(* IEC 61131-3 sources: std_i2980_v2.06_cp053/Source/IMM/ieccontrol/ODC1, 23 files *)

(* ---- ABSEInterpreter.pu ---- *)
(*
@h    ! WARNING !
@h    The Kemro K2 system (including software) only meets category B according to EN 954-1,
@h    thus it is not intended for usage in safety-relevant control applications in the field
@h    of personal safety (e.g. emergency stop).
@h    To implement potentially necessary safety-relevant control tasks, always use additional
@h    external safety devices that are intended for the particular purpose, and meet the necessary
@h    functional safety.
@h    For further information see EN 954-1 (EN ISO 13849-1) and/or the K2-x00 user manual, chapter
@h    "CE conformity, directives and standards".

*)

IMPORT_OVER_LISTFILE
 KMEM_HashMapGet
, GET_RUNTIME
, SET_WVEVENT
, cSafetyListLen
, cSEO_END
, cSEO_NOP
, cSEO_START
, cSEO_LD
, cSEO_AND
, cSEO_XOR
, cSEStackSize
, cSEC_BC_EQ_NOT
, cSEC_BC_EQ
, cSEC_BV_EQ_NOT
, cSEC_BV_EQ
, cSEC_RC_GT
, cSEC_RC_LT
, cSEC_RV_GT
, cSEC_RV_LT
, cSEC_POP
, tyMovementRegisterList
, tyODCSequenceInternal
, tsGlbSafetyData
//  tsSafetyCondition
, tySEStack
, tsODCStepPos

END_IMPORT

ALGORITHM_BLOCK ABSEInterpreter #DUMMY_EDIT_BLOCK

SYSTEM_VAR
 sv_MovementsAvailable : tyMovementRegisterList;
 sv_ODCSequenceInt : tyODCSequenceInternal;
 // sv_SafetyCondition : tsSafetyCondition;
END_VAR

SYSTEM_OBJECT
 erSEMovementNotAllowed : ALARM;
END_OBJECT

VAR_EXTERNAL
 g_SafetyData : tsGlbSafetyData;
END_VAR

VAR
 miStackPtr : INT;
 mybStack : tySEStack;
END_VAR

(*
@h    ! WARNING !
@h    The Kemro K2 system (including software) only meets category B according to EN 954-1,
@h    thus it is not intended for usage in safety-relevant control applications in the field
@h    of personal safety (e.g. emergency stop).
@h    To implement potentially necessary safety-relevant control tasks, always use additional
@h    external safety devices that are intended for the particular purpose, and meet the necessary
@h    functional safety.
@h    For further information see EN 954-1 (EN ISO 13849-1) and/or the K2-x00 user manual, chapter
@h    "CE conformity, directives and standards".

*)

FUNCTION fEvaluateCondition : BOOL
 #DUMMY_EDIT_BLOCK

VAR_INPUT
 i : DINT;
END_VAR

VAR_IN_OUT
 bResult : BOOL;
END_VAR
#BEGIN_EDIT_BLOCK
(**************************************** WARNING ********************************************
 *** The KEBA Kemro K2 System including software is not intended for safety control tasks! ***
 ***                       For further information see Comment tab!                        ***
 *********************************************************************************************)

CASE (g_SafetyData.SafetyListTmp[i].Condition) OF
    cSEC_BC_EQ_NOT:
         fEvaluateCondition := g_SafetyData.SafetyListTmp[i].pbParamBool <> EMPTY;
         IF fEvaluateCondition THEN
             bResult := g_SafetyData.SafetyListTmp[i].pbParamBool^ = FALSE;
         END_IF;

    cSEC_BC_EQ:
         fEvaluateCondition := g_SafetyData.SafetyListTmp[i].pbParamBool <> EMPTY;
         IF fEvaluateCondition THEN
             bResult := g_SafetyData.SafetyListTmp[i].pbParamBool^ = TRUE;
         END_IF;

    cSEC_BV_EQ_NOT:
         fEvaluateCondition := (g_SafetyData.SafetyListTmp[i].pbParamBool <> EMPTY)
                        AND (i < cSafetyListLen)
                        AND (g_SafetyData.SafetyListTmp[i+1].pbParamBool <> EMPTY);

         IF fEvaluateCondition THEN
             bResult := g_SafetyData.SafetyListTmp[i].pbParamBool^ <> g_SafetyData.SafetyListTmp[i+1].pbParamBool^;
         END_IF;

    cSEC_BV_EQ:
         fEvaluateCondition := (g_SafetyData.SafetyListTmp[i].pbParamBool <> EMPTY)
                        AND (i < cSafetyListLen)
                        AND (g_SafetyData.SafetyListTmp[i+1].pbParamBool <> EMPTY);

         IF fEvaluateCondition THEN
             bResult := g_SafetyData.SafetyListTmp[i].pbParamBool^ = g_SafetyData.SafetyListTmp[i+1].pbParamBool^;
         END_IF;

    cSEC_RC_GT:
         fEvaluateCondition := (g_SafetyData.SafetyListTmp[i].prParamReal <> EMPTY)
                        AND (i < cSafetyListLen);

         IF fEvaluateCondition THEN
             bResult := g_SafetyData.SafetyListTmp[i].prParamReal^ > g_SafetyData.SafetyListTmp[i+1].rValueReal;
         END_IF;

    cSEC_RC_LT:
         fEvaluateCondition := (g_SafetyData.SafetyListTmp[i].prParamReal <> EMPTY)
                        AND (i < cSafetyListLen);

         IF fEvaluateCondition THEN
             bResult := g_SafetyData.SafetyListTmp[i].prParamReal^ < g_SafetyData.SafetyListTmp[i+1].rValueReal;
         END_IF;

    cSEC_RV_GT:
         fEvaluateCondition := (g_SafetyData.SafetyListTmp[i].prParamReal <> EMPTY)
                        AND (i < cSafetyListLen)
                        AND (g_SafetyData.SafetyListTmp[i+1].prParamReal <> EMPTY);

         IF fEvaluateCondition THEN
             bResult := g_SafetyData.SafetyListTmp[i].prParamReal^ > g_SafetyData.SafetyListTmp[i+1].prParamReal^;
         END_IF;

    cSEC_RV_LT:
         fEvaluateCondition := (g_SafetyData.SafetyListTmp[i].prParamReal <> EMPTY)
                        AND (i < cSafetyListLen)
                        AND (g_SafetyData.SafetyListTmp[i+1].prParamReal <> EMPTY);

         IF fEvaluateCondition THEN
             bResult := g_SafetyData.SafetyListTmp[i].prParamReal^ < g_SafetyData.SafetyListTmp[i+1].prParamReal^;
         END_IF;

    cSEC_POP:
         IF (miStackPtr > 0) THEN
              bResult := mybStack[miStackPtr];
              miStackPtr := miStackPtr - 1;
              fEvaluateCondition := TRUE;
         END_IF;

ELSE
    fEvaluateCondition := FALSE;
END_CASE;

;#END_EDIT_BLOCK END_FUNCTION

(*
@h    ! WARNING !
@h    The Kemro K2 system (including software) only meets category B according to EN 954-1,
@h    thus it is not intended for usage in safety-relevant control applications in the field
@h    of personal safety (e.g. emergency stop).
@h    To implement potentially necessary safety-relevant control tasks, always use additional
@h    external safety devices that are intended for the particular purpose, and meet the necessary
@h    functional safety.
@h    For further information see EN 954-1 (EN ISO 13849-1) and/or the K2-x00 user manual, chapter
@h    "CE conformity, directives and standards".

*)

FUNCTION fRunSafetyCondition : BOOL
 #DUMMY_EDIT_BLOCK

VAR_INPUT
 iIdx : DINT;
END_VAR

VAR
 bValue : BOOL;
 idx : DINT;
 bResult : BOOL;
 bCondition : BOOL;
 bConditionFound : BOOL (* at least one valid condition found *);
END_VAR
#BEGIN_EDIT_BLOCK
(**************************************** WARNING ********************************************
 *** The KEBA Kemro K2 System including software is not intended for safety control tasks! ***
 ***                       For further information see Comment tab!                        ***
 *********************************************************************************************)

bValue := FALSE;
miStackPtr := -1;
idx := iIdx;

bConditionFound := FALSE;
WHILE (idx <= cSafetyListLen) DO
    CASE g_SafetyData.SafetyListTmp[idx].Operator OF
        cSEO_NOP:
            ;

        cSEO_START:
            EXIT;

        cSEO_LD:
            // each LD except first one pushes actual value to stack
            IF (miStackPtr = cSEStackSize) THEN
                bValue := FALSE; // TODO stackoverflow
            END_IF;

            miStackPtr := miStackPtr + 1;

            IF (miStackPtr > 0) THEN
               mybStack[miStackPtr] := bValue;
            END_IF;

            bResult := fEvaluateCondition(idx, bCondition);
            IF bResult THEN
               bValue := bCondition;
            END_IF;

        cSEO_AND:
            bResult := fEvaluateCondition(idx, bCondition);
            IF bResult THEN
                IF miStackPtr >= 0 THEN
                    bValue := bValue AND bCondition;
                ELSE // special case: no "LD" evaluated before, Operator should work like "LD"
                    bValue := bCondition;
                END_IF;
            END_IF;

        cSEO_OR:
            bResult := fEvaluateCondition(idx, bCondition);
            IF bResult THEN
                IF miStackPtr >= 0 THEN
                    bValue := bValue OR bCondition;
                ELSE // special case: no "LD" evaluated before, Operator should work like "LD"
                    bValue := bCondition;
                END_IF;
            END_IF;

        cSEO_XOR:
            bResult := fEvaluateCondition(idx, bCondition);
            IF bResult THEN
                IF miStackPtr >= 0 THEN
                    bValue := bValue XOR bCondition;
                ELSE // special case: no "LD" evaluated before, Operator should work like "LD"
                    bValue := bCondition;
                END_IF;
            END_IF;

        cSEO_END:
            EXIT;
    ELSE
        ; // invalid operation
    END_CASE;

    IF bResult THEN
       bConditionFound := TRUE;
    END_IF;
    idx := idx + 1;
END_WHILE;
//     dummy := Print('ABSEInterpreter.fRunSafetyCondition %s = %d',  sv_SafetyCondition.List[iIdx-1].sParameter, bValue);
fRunSafetyCondition := bValue OR (NOT bConditionFound);

;#END_EDIT_BLOCK END_FUNCTION

(*
@h    ! WARNING !
@h    The Kemro K2 system (including software) only meets category B according to EN 954-1,
@h    thus it is not intended for usage in safety-relevant control applications in the field
@h    of personal safety (e.g. emergency stop).
@h    To implement potentially necessary safety-relevant control tasks, always use additional
@h    external safety devices that are intended for the particular purpose, and meet the necessary
@h    functional safety.
@h    For further information see EN 954-1 (EN ISO 13849-1) and/or the K2-x00 user manual, chapter
@h    "CE conformity, directives and standards".

*)

FUNCTION fCheckMovement : BOOL
 #DUMMY_EDIT_BLOCK

VAR_INPUT
 StepPos : tsODCStepPos (* Step for which dependencies are checked *);
END_VAR

VAR
 i : DINT;
 bAllowed : BOOL;
 iMoveNumber : DINT;
END_VAR
#BEGIN_EDIT_BLOCK
(**************************************** WARNING ********************************************
 *** The KEBA Kemro K2 System including software is not intended for safety control tasks! ***
 ***                       For further information see Comment tab!                        ***
 *********************************************************************************************)

// DBG s:=SET_WVEVENT(1110);
bAllowed := TRUE;

IF (NOT g_SafetyData.bAvailable) THEN
    fCheckMovement := bAllowed;
    RETURN;
END_IF;

iMoveNumber := sv_ODCSequenceInt[StepPos.iColumn][StepPos.iRow].iMoveNumber;

i :=  sv_MovementsAvailable[iMoveNumber].iSESafetyProgIdx;

IF (i > 0) THEN
// DBG    s:=SET_WVEVENT(1112);
    bAllowed := fRunSafetyCondition(i);
// DBG    s:=SET_WVEVENT(1113);
    IF (NOT bAllowed) THEN
       SET_ALARM(Name := erSEMovementNotAllowed,
              SubID1 := sv_MovementsAvailable[iMoveNumber].DeviceId.CompId,
              SubID2 := sv_MovementsAvailable[iMoveNumber].DeviceId.IndexId,
              SubID3 := sv_MovementsAvailable[iMoveNumber].pMovementData^.MoveDir);

    END_IF;
    g_SafetyData.MovementAllowed[sv_MovementsAvailable[iMoveNumber].iODCSafetyMovementsEntry] := bAllowed;
END_IF;

// DBG s:=SET_WVEVENT(1114);

fCheckMovement := bAllowed;

;#END_EDIT_BLOCK END_FUNCTION

END_ALGORITHM_BLOCK

#END_OF_IEC_PART

@Puma @IecEditor 6 113 @Pou 25
@@@BEG_Comment@@@
@h    ! WARNING !
@h    The Kemro K2 system (including software) only meets category B according to EN 954-1,
@h    thus it is not intended for usage in safety-relevant control applications in the field
@h    of personal safety (e.g. emergency stop).
@h    To implement potentially necessary safety-relevant control tasks, always use additional
@h    external safety devices that are intended for the particular purpose, and meet the necessary
@h    functional safety.
@h    For further information see EN 954-1 (EN ISO 13849-1) and/or the K2-x00 user manual, chapter
@h    "CE conformity, directives and standards".

@@@END_Comment@@@

@BEG_Contents

@BEG_Func
@RT(17)FuncTreeContainer
3
@Var @RT(15)KMEM_HashMapGet @RT(0) @T @T @DERIVED 0 @F @RT(22)KEBA_STANDARD_FUNCTION @F
@T
@BEG_Attrib
0 @RT(0) @RT(0)
@END_Attrib
1 1 @F @F @F @F

@Var @RT(11)GET_RUNTIME @RT(0) @T @T @DERIVED 0 @F @RT(22)KEBA_STANDARD_FUNCTION @F
@T
@BEG_Attrib
0 @RT(0) @RT(0)
@END_Attrib
1 1 @F @F @F @F

@Var @RT(11)SET_WVEVENT @RT(0) @T @T @DERIVED 0 @F @RT(22)KEBA_STANDARD_FUNCTION @F
@T
@BEG_Attrib
0 @RT(0) @RT(0)
@END_Attrib
1 1 @F @F @F @F

@END_Func

@BEG_Const
@RT(18)ConstTreeContainer
17
@Var @RT(14)cSafetyListLen @RT(0) @T @F @DT @RT(4)DINT @RT(0) @T @T @BASIC 0 @F
@F @F
@T
@BEG_Attrib
0 @RT(3)200 @RT(39)array length of safety program variable
@END_Attrib
1 1 @F @F @F @F

@Var @RT(8)cSEO_END @RT(0) @T @F @DT @RT(4)UINT @RT(0) @T @T @BASIC 0 @F
@F @F
@T
@BEG_Attrib
0 @RT(5)16#FF @RT(14)END of program
@END_Attrib
1 1 @F @F @F @F

@Var @RT(8)cSEO_NOP @RT(0) @T @F @DT @RT(4)UINT @RT(0) @T @T @BASIC 0 @F
@F @F
@T
@BEG_Attrib
0 @RT(5)16#00 @RT(89)Operator "no operation" (e.g. line contains only additional parameter for last operation)
@END_Attrib
1 1 @F @F @F @F

@Var @RT(10)cSEO_START @RT(0) @T @F @DT @RT(4)UINT @RT(0) @T @T @BASIC 0 @F
@F @F
@T
@BEG_Attrib
0 @RT(5)16#01 @RT(92)start conditions for a certain movement defined in parameter as string (e.g. "Mold1.MoveFwd"
@END_Attrib
1 1 @F @F @F @F

@Var @RT(7)cSEO_LD @RT(0) @T @F @DT @RT(4)UINT @RT(0) @T @T @BASIC 0 @F
@F @F
@T
@BEG_Attrib
0 @RT(5)16#02 @RT(102)Load condition result, if a condition result has been calculated before this result is pushed to stack
@END_Attrib
1 1 @F @F @F @F

@Var @RT(8)cSEO_AND @RT(0) @T @F @DT @RT(4)UINT @RT(0) @T @T @BASIC 0 @F
@F @F
@T
@BEG_Attrib
0 @RT(5)16#03 @RT(53)AND operation with actual result and condition result
@END_Attrib
1 1 @F @F @F @F

@Var @RT(8)cSEO_XOR @RT(0) @T @F @DT @RT(4)UINT @RT(0) @T @T @BASIC 0 @F
@F @F
@T
@BEG_Attrib
0 @RT(5)16#05 @RT(53)XOR operation with actual result and condition result
@END_Attrib
1 1 @F @F @F @F

@Var @RT(12)cSEStackSize @RT(0) @T @F @DT @RT(3)INT @RT(0) @T @T @BASIC 0 @F
@F @F
@T
@BEG_Attrib
0 @RT(1)8 @RT(57)size of stack for condition evaluation in ABSEInterpreter
@END_Attrib
1 1 @F @F @F @F

@Var @RT(14)cSEC_BC_EQ_NOT @RT(0) @T @F @DT @RT(4)UINT @RT(0) @T @T @BASIC 0 @F
@F @F
@T
@BEG_Attrib
0 @RT(5)16#10 @RT(25)Condition BOOL SV = FALSE
@END_Attrib
1 1 @F @F @F @F

@Var @RT(10)cSEC_BC_EQ @RT(0) @T @F @DT @RT(4)UINT @RT(0) @T @T @BASIC 0 @F
@F @F
@T
@BEG_Attrib
0 @RT(5)16#11 @RT(24)Condition BOOL SV = TRUE
@END_Attrib
1 1 @F @F @F @F

@Var @RT(14)cSEC_BV_EQ_NOT @RT(0) @T @F @DT @RT(4)UINT @RT(0) @T @T @BASIC 0 @F
@F @F
@T
@BEG_Attrib
0 @RT(5)16#12 @RT(23)Condition BOOL SV <> SV
@END_Attrib
1 1 @F @F @F @F

@Var @RT(10)cSEC_BV_EQ @RT(0) @T @F @DT @RT(4)UINT @RT(0) @T @T @BASIC 0 @F
@F @F
@T
@BEG_Attrib
0 @RT(5)16#13 @RT(22)Condition BOOL SV = SV
@END_Attrib
1 1 @F @F @F @F

@Var @RT(10)cSEC_RC_GT @RT(0) @T @F @DT @RT(4)UINT @RT(0) @T @T @BASIC 0 @F
@F @F
@T
@BEG_Attrib
0 @RT(5)16#20 @RT(25)Condition REAL SV > VALUE
@END_Attrib
1 1 @F @F @F @F

@Var @RT(10)cSEC_RC_LT @RT(0) @T @F @DT @RT(4)UINT @RT(0) @T @T @BASIC 0 @F
@F @F
@T
@BEG_Attrib
0 @RT(5)16#21 @RT(25)Condition REAL SV < VALUE
@END_Attrib
1 1 @F @F @F @F

@Var @RT(10)cSEC_RV_GT @RT(0) @T @F @DT @RT(4)UINT @RT(0) @T @T @BASIC 0 @F
@F @F
@T
@BEG_Attrib
0 @RT(5)16#22 @RT(22)Condition REAL SV > SV
@END_Attrib
1 1 @F @F @F @F

@Var @RT(10)cSEC_RV_LT @RT(0) @T @F @DT @RT(4)UINT @RT(0) @T @T @BASIC 0 @F
@F @F
@T
@BEG_Attrib
0 @RT(5)16#23 @RT(22)Condition REAL SV < SV
@END_Attrib
1 1 @F @F @F @F

@Var @RT(8)cSEC_POP @RT(0) @T @F @DT @RT(4)UINT @RT(0) @T @T @BASIC 0 @F
@F @F
@T
@BEG_Attrib
0 @RT(5)16#FF @RT(24)pop Condition from Stack
@END_Attrib
1 1 @F @F @F @F

@END_Const

@BEG_Export

@BEG_Kind
@ALGORITHM_BLOCK @RT(15)ABSEInterpreter @STRUCTURED_TEXT
@RT(0) @RT(0) @RT(0)
@END_Kind

@BEG_Dcl
@RT(16)DclTreeContainer
7
@Var @RT(21)sv_MovementsAvailable @RT(0) @T @T @DERIVED 0 @T @T @DT @RT(22)tyMovementRegisterList @RT(0) @T @T @UNKNOWN 0 @F
@F @F
@T
@BEG_Attrib
3 @RT(0) @RT(0) @RT(0)
@END_Attrib
1 8 @F @F @F @F

@Var @RT(17)sv_ODCSequenceInt @RT(0) @T @T @DERIVED 0 @T @T @DT @RT(21)tyODCSequenceInternal @RT(0) @T @T @UNKNOWN 0 @F
@F @F
@T
@BEG_Attrib
3 @RT(0) @RT(0) @RT(0)
@END_Attrib
1 8 @F @F @F @F

@Var @RT(12)g_SafetyData @RT(0) @T @T @DERIVED 0 @T @T @DT @RT(15)tsGlbSafetyData @RT(0) @T @T @UNKNOWN 0 @F
@F @F
@T
@BEG_Attrib
3 @RT(0) @RT(0) @RT(0)
@END_Attrib
1 6 @F @F @F @F

@Var @RT(18)sv_SafetyCondition @RT(0) @T @T @DERIVED 0 @T @T @DT @RT(17)tsSafetyCondition @RT(0) @T @T @UNKNOWN 0 @F
@F @T
@T
@BEG_Attrib
3 @RT(0) @RT(0) @RT(0)
@END_Attrib
1 8 @F @F @F @F

@Var @RT(10)miStackPtr @RT(0) @T @F @DT @RT(3)INT @RT(0) @T @T @BASIC 0 @F
@F @F
@T
@BEG_Attrib
3 @RT(0) @RT(0) @RT(0)
@END_Attrib
1 0 @F @F @F @F

@Var @RT(8)mybStack @RT(0) @T @T @DERIVED 0 @T @T @DT @RT(9)tySEStack @RT(0) @T @T @UNKNOWN 0 @F
@F @F
@T
@BEG_Attrib
3 @RT(0) @RT(0) @RT(0)
@END_Attrib
1 0 @F @F @F @F

@Var @RT(22)erSEMovementNotAllowed @RT(0) @T @F @DT @RT(5)ALARM @RT(0) @T @T @BASIC 0 @F
@F @F
@T
@BEG_Attrib
3 @RT(0) @RT(0) @RT(0)
@END_Attrib
1 7 @F @F @F @F

@END_Dcl

@END_Export

@BEG_Body

3

@BEG_Export

@BEG_Algo
@FUNCTION @RT(18)fEvaluateCondition @STRUCTURED_TEXT
@RT(4)BOOL @RT(0) @RT(0) @F @F
@END_Algo

@BEG_Dcl
@RT(16)DclTreeContainer
2
@Var @RT(1)i @RT(0) @T @F @DT @RT(4)DINT @RT(0) @T @T @BASIC 0 @F
@F @F
@T
@BEG_Attrib
3 @RT(0) @RT(0) @RT(0)
@END_Attrib
1 1 @F @F @F @F

@Var @RT(7)bResult @RT(0) @T @F @DT @RT(4)BOOL @RT(0) @T @T @BASIC 0 @F
@F @F
@T
@BEG_Attrib
3 @RT(0) @RT(0) @RT(0)
@END_Attrib
1 2 @F @F @F @F

@END_Dcl

@END_Export

@BEG_Export

@BEG_Algo
@FUNCTION @RT(19)fRunSafetyCondition @STRUCTURED_TEXT
@RT(4)BOOL @RT(0) @RT(0) @F @F
@END_Algo

@BEG_Dcl
@RT(16)DclTreeContainer
6
@Var @RT(4)iIdx @RT(0) @T @F @DT @RT(4)DINT @RT(0) @T @T @BASIC 0 @F
@F @F
@T
@BEG_Attrib
3 @RT(0) @RT(0) @RT(0)
@END_Attrib
1 1 @F @F @F @F

@Var @RT(6)bValue @RT(0) @T @F @DT @RT(4)BOOL @RT(0) @T @T @BASIC 0 @F
@F @F
@T
@BEG_Attrib
3 @RT(0) @RT(0) @RT(0)
@END_Attrib
1 0 @F @F @F @F

@Var @RT(3)idx @RT(0) @T @F @DT @RT(4)DINT @RT(0) @T @T @BASIC 0 @F
@F @F
@T
@BEG_Attrib
3 @RT(0) @RT(0) @RT(0)
@END_Attrib
1 0 @F @F @F @F

@Var @RT(7)bResult @RT(0) @T @F @DT @RT(4)BOOL @RT(0) @T @T @BASIC 0 @F
@F @F
@T
@BEG_Attrib
3 @RT(0) @RT(0) @RT(0)
@END_Attrib
1 0 @F @F @F @F

@Var @RT(10)bCondition @RT(0) @T @F @DT @RT(4)BOOL @RT(0) @T @T @BASIC 0 @F
@F @F
@T
@BEG_Attrib
3 @RT(0) @RT(0) @RT(0)
@END_Attrib
1 0 @F @F @F @F

@Var @RT(15)bConditionFound @RT(0) @T @F @DT @RT(4)BOOL @RT(0) @T @T @BASIC 0 @F
@F @F
@T
@BEG_Attrib
3 @RT(0) @RT(34)at least one valid condition found @RT(0)
@END_Attrib
1 0 @F @F @F @F

@END_Dcl

@END_Export

@BEG_Export

@BEG_Algo
@FUNCTION @RT(14)fCheckMovement @STRUCTURED_TEXT
@RT(4)BOOL @RT(0) @RT(0) @F @F
@END_Algo

@BEG_Dcl
@RT(16)DclTreeContainer
4
@Var @RT(7)StepPos @RT(0) @T @T @DERIVED 0 @T @T @DT @RT(12)tsODCStepPos @RT(0) @T @T @UNKNOWN 0 @F
@F @F
@T
@BEG_Attrib
3 @RT(0) @RT(39)Step for which dependencies are checked @RT(0)
@END_Attrib
1 1 @F @F @F @F

@Var @RT(1)i @RT(0) @T @F @DT @RT(4)DINT @RT(0) @T @T @BASIC 0 @F
@F @F
@T
@BEG_Attrib
3 @RT(0) @RT(0) @RT(0)
@END_Attrib
1 0 @F @F @F @F

@Var @RT(8)bAllowed @RT(0) @T @F @DT @RT(4)BOOL @RT(0) @T @T @BASIC 0 @F
@F @F
@T
@BEG_Attrib
3 @RT(0) @RT(0) @RT(0)
@END_Attrib
1 0 @F @F @F @F

@Var @RT(11)iMoveNumber @RT(0) @T @F @DT @RT(4)DINT @RT(0) @T @T @BASIC 0 @F
@F @F
@T
@BEG_Attrib
3 @RT(0) @RT(0) @RT(0)
@END_Attrib
1 0 @F @F @F @F

@END_Dcl

@END_Export

@BEG_Body
@TL(86)
(**************************************** WARNING ********************************************
 *** The KEBA Kemro K2 System including software is not intended for safety control tasks! ***
 ***                       For further information see Comment tab!                        ***
 *********************************************************************************************)

CASE (g_SafetyData.SafetyListTmp[i].Condition) OF
    cSEC_BC_EQ_NOT:
         fEvaluateCondition := g_SafetyData.SafetyListTmp[i].pbParamBool <> EMPTY;
         IF fEvaluateCondition THEN
             bResult := g_SafetyData.SafetyListTmp[i].pbParamBool^ = FALSE;
         END_IF;

    cSEC_BC_EQ:
         fEvaluateCondition := g_SafetyData.SafetyListTmp[i].pbParamBool <> EMPTY;
         IF fEvaluateCondition THEN
             bResult := g_SafetyData.SafetyListTmp[i].pbParamBool^ = TRUE;
         END_IF;

    cSEC_BV_EQ_NOT:
         fEvaluateCondition := (g_SafetyData.SafetyListTmp[i].pbParamBool <> EMPTY)
                        AND (i < cSafetyListLen)
                        AND (g_SafetyData.SafetyListTmp[i+1].pbParamBool <> EMPTY);

         IF fEvaluateCondition THEN
             bResult := g_SafetyData.SafetyListTmp[i].pbParamBool^ <> g_SafetyData.SafetyListTmp[i+1].pbParamBool^;
         END_IF;

    cSEC_BV_EQ:
         fEvaluateCondition := (g_SafetyData.SafetyListTmp[i].pbParamBool <> EMPTY)
                        AND (i < cSafetyListLen)
                        AND (g_SafetyData.SafetyListTmp[i+1].pbParamBool <> EMPTY);

         IF fEvaluateCondition THEN
             bResult := g_SafetyData.SafetyListTmp[i].pbParamBool^ = g_SafetyData.SafetyListTmp[i+1].pbParamBool^;
         END_IF;

    cSEC_RC_GT:
         fEvaluateCondition := (g_SafetyData.SafetyListTmp[i].prParamReal <> EMPTY)
                        AND (i < cSafetyListLen);

         IF fEvaluateCondition THEN
             bResult := g_SafetyData.SafetyListTmp[i].prParamReal^ > g_SafetyData.SafetyListTmp[i+1].rValueReal;
         END_IF;

    cSEC_RC_LT:
         fEvaluateCondition := (g_SafetyData.SafetyListTmp[i].prParamReal <> EMPTY)
                        AND (i < cSafetyListLen);

         IF fEvaluateCondition THEN
             bResult := g_SafetyData.SafetyListTmp[i].prParamReal^ < g_SafetyData.SafetyListTmp[i+1].rValueReal;
         END_IF;

    cSEC_RV_GT:
         fEvaluateCondition := (g_SafetyData.SafetyListTmp[i].prParamReal <> EMPTY)
                        AND (i < cSafetyListLen)
                        AND (g_SafetyData.SafetyListTmp[i+1].prParamReal <> EMPTY);

         IF fEvaluateCondition THEN
             bResult := g_SafetyData.SafetyListTmp[i].prParamReal^ > g_SafetyData.SafetyListTmp[i+1].prParamReal^;
         END_IF;

    cSEC_RV_LT:
         fEvaluateCondition := (g_SafetyData.SafetyListTmp[i].prParamReal <> EMPTY)
                        AND (i < cSafetyListLen)
                        AND (g_SafetyData.SafetyListTmp[i+1].prParamReal <> EMPTY);

         IF fEvaluateCondition THEN
             bResult := g_SafetyData.SafetyListTmp[i].prParamReal^ < g_SafetyData.SafetyListTmp[i+1].prParamReal^;
         END_IF;

    cSEC_POP:
         IF (miStackPtr > 0) THEN
              bResult := mybStack[miStackPtr];
              miStackPtr := miStackPtr - 1;
              fEvaluateCondition := TRUE;
         END_IF;

ELSE
    fEvaluateCondition := FALSE;
END_CASE;

@END_Body

@@@BEG_Comment@@@
@TL(12)
@h    ! WARNING !
@h    The Kemro K2 system (including software) only meets category B according to EN 954-1,
@h    thus it is not intended for usage in safety-relevant control applications in the field
@h    of personal safety (e.g. emergency stop).
@h    To implement potentially necessary safety-relevant control tasks, always use additional
@h    external safety devices that are intended for the particular purpose, and meet the necessary
@h    functional safety.
@h    For further information see EN 954-1 (EN ISO 13849-1) and/or the K2-x00 user manual, chapter
@h    "CE conformity, directives and standards".

@@@END_Comment@@@

@BEG_Body
@TL(84)
(**************************************** WARNING ********************************************
 *** The KEBA Kemro K2 System including software is not intended for safety control tasks! ***
 ***                       For further information see Comment tab!                        ***
 *********************************************************************************************)

bValue := FALSE;
miStackPtr := -1;
idx := iIdx;

bConditionFound := FALSE;
WHILE (idx <= cSafetyListLen) DO
    CASE g_SafetyData.SafetyListTmp[idx].Operator OF
        cSEO_NOP:
            ;

        cSEO_START:
            EXIT;

        cSEO_LD:
            // each LD except first one pushes actual value to stack
            IF (miStackPtr = cSEStackSize) THEN
                bValue := FALSE; // TODO stackoverflow
            END_IF;

            miStackPtr := miStackPtr + 1;

            IF (miStackPtr > 0) THEN
               mybStack[miStackPtr] := bValue;
            END_IF;

            bResult := fEvaluateCondition(idx, bCondition);
            IF bResult THEN
               bValue := bCondition;
            END_IF;

        cSEO_AND:
            bResult := fEvaluateCondition(idx, bCondition);
            IF bResult THEN
                IF miStackPtr >= 0 THEN
                    bValue := bValue AND bCondition;
                ELSE // special case: no "LD" evaluated before, Operator should work like "LD"
                    bValue := bCondition;
                END_IF;
            END_IF;

        cSEO_OR:
            bResult := fEvaluateCondition(idx, bCondition);
            IF bResult THEN
                IF miStackPtr >= 0 THEN
                    bValue := bValue OR bCondition;
                ELSE // special case: no "LD" evaluated before, Operator should work like "LD"
                    bValue := bCondition;
                END_IF;
            END_IF;

        cSEO_XOR:
            bResult := fEvaluateCondition(idx, bCondition);
            IF bResult THEN
                IF miStackPtr >= 0 THEN
                    bValue := bValue XOR bCondition;
                ELSE // special case: no "LD" evaluated before, Operator should work like "LD"
                    bValue := bCondition;
                END_IF;
            END_IF;

        cSEO_END:
            EXIT;
    ELSE
        ; // invalid operation
    END_CASE;

    IF bResult THEN
       bConditionFound := TRUE;
    END_IF;
    idx := idx + 1;
END_WHILE;
//     dummy := Print('ABSEInterpreter.fRunSafetyCondition %s = %d',  sv_SafetyCondition.List[iIdx-1].sParameter, bValue);
fRunSafetyCondition := bValue OR (NOT bConditionFound);

@END_Body

@@@BEG_Comment@@@
@TL(12)
@h    ! WARNING !
@h    The Kemro K2 system (including software) only meets category B according to EN 954-1,
@h    thus it is not intended for usage in safety-relevant control applications in the field
@h    of personal safety (e.g. emergency stop).
@h    To implement potentially necessary safety-relevant control tasks, always use additional
@h    external safety devices that are intended for the particular purpose, and meet the necessary
@h    functional safety.
@h    For further information see EN 954-1 (EN ISO 13849-1) and/or the K2-x00 user manual, chapter
@h    "CE conformity, directives and standards".

@@@END_Comment@@@

@BEG_Body
@TL(36)
(**************************************** WARNING ********************************************
 *** The KEBA Kemro K2 System including software is not intended for safety control tasks! ***
 ***                       For further information see Comment tab!                        ***
 *********************************************************************************************)

// DBG s:=SET_WVEVENT(1110);
bAllowed := TRUE;

IF (NOT g_SafetyData.bAvailable) THEN
    fCheckMovement := bAllowed;
    RETURN;
END_IF;

iMoveNumber := sv_ODCSequenceInt[StepPos.iColumn][StepPos.iRow].iMoveNumber;

i :=  sv_MovementsAvailable[iMoveNumber].iSESafetyProgIdx;

IF (i > 0) THEN
// DBG    s:=SET_WVEVENT(1112);
    bAllowed := fRunSafetyCondition(i);
// DBG    s:=SET_WVEVENT(1113);
    IF (NOT bAllowed) THEN
       SET_ALARM(Name := erSEMovementNotAllowed,
              SubID1 := sv_MovementsAvailable[iMoveNumber].DeviceId.CompId,
              SubID2 := sv_MovementsAvailable[iMoveNumber].DeviceId.IndexId,
              SubID3 := sv_MovementsAvailable[iMoveNumber].pMovementData^.MoveDir);

    END_IF;
    g_SafetyData.MovementAllowed[sv_MovementsAvailable[iMoveNumber].iODCSafetyMovementsEntry] := bAllowed;
END_IF;

// DBG s:=SET_WVEVENT(1114);

fCheckMovement := bAllowed;

@END_Body

@@@BEG_Comment@@@
@TL(12)
@h    ! WARNING !
@h    The Kemro K2 system (including software) only meets category B according to EN 954-1,
@h    thus it is not intended for usage in safety-relevant control applications in the field
@h    of personal safety (e.g. emergency stop).
@h    To implement potentially necessary safety-relevant control tasks, always use additional
@h    external safety devices that are intended for the particular purpose, and meet the necessary
@h    functional safety.
@h    For further information see EN 954-1 (EN ISO 13849-1) and/or the K2-x00 user manual, chapter
@h    "CE conformity, directives and standards".

@@@END_Comment@@@
@END_Body

@END_Contents

(* ---- FCreateODCVersion.pu ---- *)
(*
@h    ! WARNING !
@h    The Kemro K2 system (including software) only meets category B according to EN 954-1,
@h    thus it is not intended for usage in safety-relevant control applications in the field
@h    of personal safety (e.g. emergency stop).
@h    To implement potentially necessary safety-relevant control tasks, always use additional
@h    external safety devices that are intended for the particular purpose, and meet the necessary
@h    functional safety.
@h    For further information see EN 954-1 (EN ISO 13849-1) and/or the K2-x00 user manual, chapter
@h    "CE conformity, directives and standards".

this file is automatically created by clearcase makebaseline
and contains versioninformation of component
*)

IMPORT_OVER_LISTFILE
 FWriteComponentVersion

END_IMPORT

FUNCTION FCreateODCVersion : BOOL #DUMMY_EDIT_BLOCK

VAR CONSTANT
 sComponentName : STRING(255) := 'ApplMoldMachineODC';
 iComponentNumber : DINT := 6735;
 sVersionString : STRING(255) := 'ApplMoldMachineODC_01.36';
 iVersionMajor : DINT := 1;
 iVersionMinor : DINT := 36;
END_VAR
#BEGIN_EDIT_BLOCK
(**************************************** WARNING ********************************************
 *** The KEBA Kemro K2 System including software is not intended for safety control tasks! ***
 ***                       For further information see Comment tab!                        ***
 *********************************************************************************************)

FCreateODCVersion := FWriteComponentVersion(
        sComponentName,
        iComponentNumber,
        sVersionString,
        iVersionMajor,
        iVersionMinor
);

;#END_EDIT_BLOCK END_FUNCTION

#END_OF_IEC_PART

@Puma @IecEditor 6 68 @Pou 25
@@@BEG_Comment@@@
@h    ! WARNING !
@h    The Kemro K2 system (including software) only meets category B according to EN 954-1,
@h    thus it is not intended for usage in safety-relevant control applications in the field
@h    of personal safety (e.g. emergency stop).
@h    To implement potentially necessary safety-relevant control tasks, always use additional
@h    external safety devices that are intended for the particular purpose, and meet the necessary
@h    functional safety.
@h    For further information see EN 954-1 (EN ISO 13849-1) and/or the K2-x00 user manual, chapter
@h    "CE conformity, directives and standards".

this file is automatically created by clearcase makebaseline
and contains versioninformation of component
@@@END_Comment@@@

@BEG_Contents

@BEG_Func
@RT(17)FuncTreeContainer
1
@Var @RT(22)FWriteComponentVersion @RT(0) @T @F @DT @RT(0) @RT(0) @T @T @UNKNOWN 0 @F
@F @F
@T
@BEG_Attrib
0 @RT(0) @RT(0)
@END_Attrib
1 1 @F @F @F @F

@END_Func

@BEG_Const
@RT(18)ConstTreeContainer
0
@END_Const

@BEG_Export

@BEG_Kind
@FUNCTION @RT(17)FCreateODCVersion @STRUCTURED_TEXT
@RT(4)BOOL @RT(0) @RT(0)
@END_Kind

@BEG_Dcl
@RT(16)DclTreeContainer
5
@Var @RT(14)sComponentName @RT(0) @T @F @DT @RT(11)STRING(255) @RT(0) @T @T @STRING 0 @F @RT(3)255 @F
@F @F
@T
@BEG_Attrib
3 @RT(20)'ApplMoldMachineODC' @RT(0) @RT(0)
@END_Attrib
1 15 @F @F @F @F

@Var @RT(16)iComponentNumber @RT(0) @T @F @DT @RT(4)DINT @RT(0) @T @T @BASIC 0 @F
@F @F
@T
@BEG_Attrib
3 @RT(4)6735 @RT(0) @RT(0)
@END_Attrib
1 15 @F @F @F @F

@Var @RT(14)sVersionString @RT(0) @T @F @DT @RT(11)STRING(255) @RT(0) @T @T @STRING 0 @F @RT(3)255 @F
@F @F
@T
@BEG_Attrib
3 @RT(26)'ApplMoldMachineODC_01.36' @RT(0) @RT(0)
@END_Attrib
1 15 @F @F @F @F

@Var @RT(13)iVersionMajor @RT(0) @T @F @DT @RT(4)DINT @RT(0) @T @T @BASIC 0 @F
@F @F
@T
@BEG_Attrib
3 @RT(1)1 @RT(0) @RT(0)
@END_Attrib
1 15 @F @F @F @F

@Var @RT(13)iVersionMinor @RT(0) @T @F @DT @RT(4)DINT @RT(0) @T @T @BASIC 0 @F
@F @F
@T
@BEG_Attrib
3 @RT(2)36 @RT(0) @RT(0)
@END_Attrib
1 15 @F @F @F @F

@END_Dcl

@END_Export

@BEG_Body
@TL(13)
(**************************************** WARNING ********************************************
 *** The KEBA Kemro K2 System including software is not intended for safety control tasks! ***
 ***                       For further information see Comment tab!                        ***
 *********************************************************************************************)

FCreateODCVersion := FWriteComponentVersion(
        sComponentName,
        iComponentNumber,
        sVersionString,
        iVersionMajor,
        iVersionMinor
);

@END_Body

@END_Contents

(* ---- FSEMoveIDToValue.pu ---- *)
(*
@h    ! WARNING !
@h    The Kemro K2 system (including software) only meets category B according to EN 954-1,
@h    thus it is not intended for usage in safety-relevant control applications in the field
@h    of personal safety (e.g. emergency stop).
@h    To implement potentially necessary safety-relevant control tasks, always use additional
@h    external safety devices that are intended for the particular purpose, and meet the necessary
@h    functional safety.
@h    For further information see EN 954-1 (EN ISO 13849-1) and/or the K2-x00 user manual, chapter
@h    "CE conformity, directives and standards".

"<FU>.<string movedir>" -> "<FU>.<integer movedir>"
e.g. "Mold1.MoveFwd" -> "Mold1.12"

returns true if no error

*)

IMPORT_OVER_LISTFILE
 cMoveFwd
, cMoveBwd

END_IMPORT

FUNCTION FSEMoveIDToValue : BOOL #DUMMY_EDIT_BLOCK

VAR_IN_OUT
 s : STRING(255) (* movedir definition to be converted *);
END_VAR

VAR
 i : DINT;
 sTmpString : STRING(15);
END_VAR
#BEGIN_EDIT_BLOCK
(**************************************** WARNING ********************************************
 *** The KEBA Kemro K2 System including software is not intended for safety control tasks! ***
 ***                       For further information see Comment tab!                        ***
 *********************************************************************************************)

FSEMoveIDToValue := FALSE;

i := FIND(s, ".");

IF (i = 0) THEN
    RETURN;
END_IF;

sTmpString := RIGHT(s, LEN(s) - i);
s := LEFT(s, i);

IF (sTmpString = "MoveBwd") THEN
    i := cMoveBwd;
ELSIF (sTmpString = "MoveFwd") THEN
    i := cMoveFwd;
ELSE
    RETURN;
END_IF;

s := CONCAT(s, DINT_TO_STRING(i));
FSEMoveIDToValue := TRUE;

;#END_EDIT_BLOCK END_FUNCTION

#END_OF_IEC_PART

@Puma @IecEditor 6 113 @Pou 25
@@@BEG_Comment@@@
@h    ! WARNING !
@h    The Kemro K2 system (including software) only meets category B according to EN 954-1,
@h    thus it is not intended for usage in safety-relevant control applications in the field
@h    of personal safety (e.g. emergency stop).
@h    To implement potentially necessary safety-relevant control tasks, always use additional
@h    external safety devices that are intended for the particular purpose, and meet the necessary
@h    functional safety.
@h    For further information see EN 954-1 (EN ISO 13849-1) and/or the K2-x00 user manual, chapter
@h    "CE conformity, directives and standards".

"<FU>.<string movedir>" -> "<FU>.<integer movedir>"
e.g. "Mold1.MoveFwd" -> "Mold1.12"

returns true if no error

@@@END_Comment@@@

@BEG_Contents

@BEG_Func
@RT(17)FuncTreeContainer
0
@END_Func

@BEG_Const
@RT(18)ConstTreeContainer
2
@Var @RT(8)cMoveFwd @RT(0) @T @F @DT @RT(4)DINT @RT(0) @T @T @BASIC 0 @F
@F @F
@T
@BEG_Attrib
0 @RT(2)12 @RT(16)movement forward
@END_Attrib
1 1 @F @F @F @F

@Var @RT(8)cMoveBwd @RT(0) @T @F @DT @RT(4)DINT @RT(0) @T @T @BASIC 0 @F
@F @F
@T
@BEG_Attrib
0 @RT(2)11 @RT(17)movement backward
@END_Attrib
1 1 @F @F @F @F

@END_Const

@BEG_Export

@BEG_Kind
@FUNCTION @RT(16)FSEMoveIDToValue @STRUCTURED_TEXT
@RT(4)BOOL @RT(0) @RT(0)
@END_Kind

@BEG_Dcl
@RT(16)DclTreeContainer
3
@Var @RT(1)s @RT(0) @T @F @DT @RT(11)STRING(255) @RT(0) @T @T @STRING 0 @F @RT(3)255 @F
@F @F
@T
@BEG_Attrib
3 @RT(0) @RT(34)movedir definition to be converted @RT(0)
@END_Attrib
1 2 @F @F @F @F

@Var @RT(1)i @RT(0) @T @F @DT @RT(4)DINT @RT(0) @T @T @BASIC 0 @F
@F @F
@T
@BEG_Attrib
3 @RT(0) @RT(0) @RT(0)
@END_Attrib
1 0 @F @F @F @F

@Var @RT(10)sTmpString @RT(0) @T @F @DT @RT(10)STRING(15) @RT(0) @T @T @STRING 0 @F @RT(2)15 @F
@F @F
@T
@BEG_Attrib
3 @RT(0) @RT(0) @RT(0)
@END_Attrib
1 0 @F @F @F @F

@END_Dcl

@END_Export

@BEG_Body
@TL(28)
(**************************************** WARNING ********************************************
 *** The KEBA Kemro K2 System including software is not intended for safety control tasks! ***
 ***                       For further information see Comment tab!                        ***
 *********************************************************************************************)

FSEMoveIDToValue := FALSE;

i := FIND(s, ".");

IF (i = 0) THEN
    RETURN;
END_IF;

sTmpString := RIGHT(s, LEN(s) - i);
s := LEFT(s, i);

IF (sTmpString = "MoveBwd") THEN
    i := cMoveBwd;
ELSIF (sTmpString = "MoveFwd") THEN
    i := cMoveFwd;
ELSE
    RETURN;
END_IF;

s := CONCAT(s, DINT_TO_STRING(i));
FSEMoveIDToValue := TRUE;

@END_Body

@END_Contents

(* ---- FBAddDependency.pu ---- *)
IMPORT_OVER_LISTFILE
 tyODCDependencyArray
, tsODCDeviceMovementList
, tyMovementRegisterList

END_IMPORT

FUNCTION_BLOCK FBAddDependency #DUMMY_EDIT_BLOCK

VAR_INPUT
 iFuIndex : DINT (* index in sv_ODCDeviceMovements *);
 iMoveNr : DINT (* 0: not safety relevant, >0: movement number *);
 iCount : DINT;
 iMode : DINT (* 0: replace existing dependency 1: add condition to actual dependency  *);
END_VAR

VAR_IN_OUT
 Dependency : tyODCDependencyArray (* actual step dependency *);
END_VAR

SYSTEM_VAR
 sv_ODCDeviceMovements : tsODCDeviceMovementList (* list of all devices that registered movements for the ODC *);
 sv_MovementsAvailable : tyMovementRegisterList;
END_VAR

VAR_TEMP
 i : DINT;
 k : DINT;
END_VAR

VAR
 tmpDependency : LWORD;
 iInstanceableMovement : DINT;
 iBitNumber : DINT;
END_VAR
#BEGIN_EDIT_BLOCK
(**************************************** WARNING ********************************************
 *** The KEBA Kemro K2 System including software is not intended for safety control tasks! ***
 ***                       For further information see Comment tab!                        ***
 *********************************************************************************************)

IF iMoveNr <= 0 THEN
   Dependency[iFuIndex].Dependency := cNoDependency;
ELSE
   //get movement number in sv_ODCDeviceMovements
   FOR i := 1 TO sv_ODCDeviceMovements.Devices[iFuIndex].iNumberOfMovements DO

      IF sv_ODCDeviceMovements.Devices[iFuIndex].Movements[i]^ = sv_MovementsAvailable[iMoveNr].pMovementData^ THEN
         //move number found -> set the according bit
         tmpDependency := cFirstBit;

         //first movement: shift right 0, second movement: shift right 1, ...
         tmpDependency := SHR(tmpDependency, (i-1));

         IF iMode = 0 THEN
            //replace dependency
            Dependency[iFuIndex].Dependency := tmpDependency;
         ELSE
            //add dependency
            Dependency[iFuIndex].Dependency := Dependency[iFuIndex].Dependency OR tmpDependency;
         END_IF;

         //check if it is an instanceable movement and set correct bit
         IF sv_ODCDeviceMovements.Devices[iFuIndex].Movements[i]^.bInstanceable THEN
            tmpDependency := cFirstBit;

            //first instanceable movement: bit 21-30, second instanceable movement: bit 31-40
            //third instanceable movement: bit 41-50, fourth instanceable movement: bit 51-60

            //find out if it is the first, second, third or fourth instanceable movement in this function unit
            iInstanceableMovement := 1;
            FOR k := 1 TO cMaxSRInstanceableMovements DO
               IF i = sv_ODCDeviceMovements.Devices[iFuIndex].InstanceableMovements[k] THEN
                  iInstanceableMovement := k;
                  EXIT;
               END_IF;
            END_FOR;

            iBitNumber := cMaxDeviceMovements + ((iInstanceableMovement - 1) * cMaxIntermediateConditions) + iCount - 1;
            tmpDependency := SHR(tmpDependency, iBitNumber);

            //mode must not be checked here
            Dependency[iFuIndex].Dependency := Dependency[iFuIndex].Dependency OR tmpDependency;
         END_IF;

         EXIT;
      END_IF;
   END_FOR;
END_IF;

;#END_EDIT_BLOCK END_FUNCTION_BLOCK

#END_OF_IEC_PART

@Puma @IecEditor 6 127 @Pou 25
@@@BEG_Comment@@@

@@@END_Comment@@@

@BEG_Contents

@BEG_Func
@RT(17)FuncTreeContainer
0
@END_Func

@BEG_Const
@RT(18)ConstTreeContainer
0
@END_Const

@BEG_Export

@BEG_Kind
@FUNCTION_BLOCK @RT(15)FBAddDependency @STRUCTURED_TEXT
@RT(0) @RT(0) @RT(0)
@END_Kind

@BEG_Dcl
@RT(16)DclTreeContainer
12
@Var @RT(8)iFuIndex @RT(0) @T @F @DT @RT(4)DINT @RT(0) @T @T @BASIC 0 @F
@F @F
@T
@BEG_Attrib
3 @RT(0) @RT(30)index in sv_ODCDeviceMovements @RT(0)
@END_Attrib
1 1 @F @F @F @F

@Var @RT(7)iMoveNr @RT(0) @T @F @DT @RT(4)DINT @RT(0) @T @T @BASIC 0 @F
@F @F
@T
@BEG_Attrib
3 @RT(0) @RT(43)0: not safety relevant, >0: movement number @RT(0)
@END_Attrib
1 1 @F @F @F @F

@Var @RT(6)iCount @RT(0) @T @F @DT @RT(4)DINT @RT(0) @T @T @BASIC 0 @F
@F @F
@T
@BEG_Attrib
3 @RT(0) @RT(0) @RT(0)
@END_Attrib
1 1 @F @F @F @F

@Var @RT(5)iMode @RT(0) @T @F @DT @RT(4)DINT @RT(0) @T @T @BASIC 0 @F
@F @F
@T
@BEG_Attrib
3 @RT(0) @RT(69)0: replace existing dependency 1: add condition to actual dependency  @RT(0)
@END_Attrib
1 1 @F @F @F @F

@Var @RT(10)Dependency @RT(0) @T @T @DERIVED 0 @T @T @DT @RT(20)tyODCDependencyArray @RT(0) @T @T @UNKNOWN 0 @F
@F @F
@T
@BEG_Attrib
3 @RT(0) @RT(22)actual step dependency @RT(0)
@END_Attrib
1 2 @F @F @F @F

@Var @RT(1)i @RT(0) @T @F @DT @RT(4)DINT @RT(0) @T @T @BASIC 0 @F
@F @F
@T
@BEG_Attrib
3 @RT(0) @RT(0) @RT(0)
@END_Attrib
1 4 @F @F @F @F

@Var @RT(13)tmpDependency @RT(0) @T @F @DT @RT(5)LWORD @RT(0) @T @T @BASIC 0 @F
@F @F
@T
@BEG_Attrib
3 @RT(0) @RT(0) @RT(0)
@END_Attrib
1 0 @F @F @F @F

@Var @RT(21)sv_ODCDeviceMovements @RT(0) @T @T @DERIVED 0 @T @T @DT @RT(23)tsODCDeviceMovementList @RT(0) @T @T @UNKNOWN 0 @F
@F @F
@T
@BEG_Attrib
3 @RT(0) @RT(57)list of all devices that registered movements for the ODC @RT(0)
@END_Attrib
1 8 @F @F @F @F

@Var @RT(21)sv_MovementsAvailable @RT(0) @T @T @DERIVED 0 @T @T @DT @RT(22)tyMovementRegisterList @RT(0) @T @T @UNKNOWN 0 @F
@F @F
@T
@BEG_Attrib
3 @RT(0) @RT(0) @RT(0)
@END_Attrib
1 8 @F @F @F @F

@Var @RT(1)k @RT(0) @T @F @DT @RT(4)DINT @RT(0) @T @T @BASIC 0 @F
@F @F
@T
@BEG_Attrib
3 @RT(0) @RT(0) @RT(0)
@END_Attrib
1 4 @F @F @F @F

@Var @RT(21)iInstanceableMovement @RT(0) @T @F @DT @RT(4)DINT @RT(0) @T @T @BASIC 0 @F
@F @F
@T
@BEG_Attrib
3 @RT(0) @RT(0) @RT(0)
@END_Attrib
1 0 @F @F @F @F

@Var @RT(10)iBitNumber @RT(0) @T @F @DT @RT(4)DINT @RT(0) @T @T @BASIC 0 @F
@F @F
@T
@BEG_Attrib
3 @RT(0) @RT(0) @RT(0)
@END_Attrib
1 0 @F @F @F @F

@END_Dcl

@END_Export

@BEG_Body
@TL(54)
(**************************************** WARNING ********************************************
 *** The KEBA Kemro K2 System including software is not intended for safety control tasks! ***
 ***                       For further information see Comment tab!                        ***
 *********************************************************************************************)

IF iMoveNr <= 0 THEN
   Dependency[iFuIndex].Dependency := cNoDependency;
ELSE
   //get movement number in sv_ODCDeviceMovements
   FOR i := 1 TO sv_ODCDeviceMovements.Devices[iFuIndex].iNumberOfMovements DO

      IF sv_ODCDeviceMovements.Devices[iFuIndex].Movements[i]^ = sv_MovementsAvailable[iMoveNr].pMovementData^ THEN
         //move number found -> set the according bit
         tmpDependency := cFirstBit;

         //first movement: shift right 0, second movement: shift right 1, ...
         tmpDependency := SHR(tmpDependency, (i-1));

         IF iMode = 0 THEN
            //replace dependency
            Dependency[iFuIndex].Dependency := tmpDependency;
         ELSE
            //add dependency
            Dependency[iFuIndex].Dependency := Dependency[iFuIndex].Dependency OR tmpDependency;
         END_IF;

         //check if it is an instanceable movement and set correct bit
         IF sv_ODCDeviceMovements.Devices[iFuIndex].Movements[i]^.bInstanceable THEN
            tmpDependency := cFirstBit;

            //first instanceable movement: bit 21-30, second instanceable movement: bit 31-40
            //third instanceable movement: bit 41-50, fourth instanceable movement: bit 51-60

            //find out if it is the first, second, third or fourth instanceable movement in this function unit
            iInstanceableMovement := 1;
            FOR k := 1 TO cMaxSRInstanceableMovements DO
               IF i = sv_ODCDeviceMovements.Devices[iFuIndex].InstanceableMovements[k] THEN
                  iInstanceableMovement := k;
                  EXIT;
               END_IF;
            END_FOR;

            iBitNumber := cMaxDeviceMovements + ((iInstanceableMovement - 1) * cMaxIntermediateConditions) + iCount - 1;
            tmpDependency := SHR(tmpDependency, iBitNumber);

            //mode must not be checked here
            Dependency[iFuIndex].Dependency := Dependency[iFuIndex].Dependency OR tmpDependency;
         END_IF;

         EXIT;
      END_IF;
   END_FOR;
END_IF;

@END_Body

@END_Contents

(* ---- FBInterpreterCheckIsRightJoin.pu ---- *)
(*
@h    ! WARNING !
@h    The Kemro K2 system (including software) only meets category B according to EN 954-1,
@h    thus it is not intended for usage in safety-relevant control applications in the field
@h    of personal safety (e.g. emergency stop).
@h    To implement potentially necessary safety-relevant control tasks, always use additional
@h    external safety devices that are intended for the particular purpose, and meet the necessary
@h    functional safety.
@h    For further information see EN 954-1 (EN ISO 13849-1) and/or the K2-x00 user manual, chapter
@h    "CE conformity, directives and standards".

Helper for FBInterpreterFindEndOfParalle.pu
Check if we have a join on iLine where the leftmost column with a EndParallel
is iColumnStartBranch
-> this is used to find the end of a parallel branch
*)

IMPORT_OVER_LISTFILE
 cMoveEndParallel
, KODC_Sequence
, FBDebugTrace2

END_IMPORT

FUNCTION_BLOCK FBInterpreterCheckIsRightJoin #DUMMY_EDIT_BLOCK

VAR_IN_OUT
 odcSequence : KODC_Sequence (* [col][line] *);
END_VAR

VAR_INPUT
 iColumnStartBranch : DINT;
 iLine : DINT;
END_VAR

VAR_OUTPUT
 bIsJoin : BOOL;
 bError : BOOL;
END_VAR

VAR_TEMP
 iTmpColumn : DINT;
END_VAR

VAR
 fbDebugTrace2 : FBDebugTrace2;
END_VAR
#BEGIN_EDIT_BLOCK
bError := FALSE;
bIsJoin := FALSE;

FOR iTmpColumn := 1 TO cMaxParallelMovements DO
   IF odcSequence[iTmpColumn][iLine].iMoveId = cMoveEndParallel THEN
      IF iTmpColumn < iColumnStartBranch THEN
         fbDebugTrace2(nODCInterpreter, 'found a EndPParallel at pos:x/x, that tries to join to the wrong parent branch');
         bError := TRUE;
         RETURN; (* error tried to join to somewhere else
                  before we got our wanted join *)
      END_IF;
      IF iTmpColumn = iColumnStartBranch THEN
         (* found where this branch joins again with iColumn *)
         bIsJoin := TRUE;
         RETURN;
      END_IF;
      (* otherwise something else tries to join into this column from the right side
         this is OK, ignore it *)
   END_IF;
END_FOR;

;#END_EDIT_BLOCK END_FUNCTION_BLOCK

#END_OF_IEC_PART

@Puma @IecEditor 6 95 @Pou 25
@@@BEG_Comment@@@
@h    ! WARNING !
@h    The Kemro K2 system (including software) only meets category B according to EN 954-1,
@h    thus it is not intended for usage in safety-relevant control applications in the field
@h    of personal safety (e.g. emergency stop).
@h    To implement potentially necessary safety-relevant control tasks, always use additional
@h    external safety devices that are intended for the particular purpose, and meet the necessary
@h    functional safety.
@h    For further information see EN 954-1 (EN ISO 13849-1) and/or the K2-x00 user manual, chapter
@h    "CE conformity, directives and standards".

Helper for FBInterpreterFindEndOfParalle.pu
Check if we have a join on iLine where the leftmost column with a EndParallel
is iColumnStartBranch
-> this is used to find the end of a parallel branch
@@@END_Comment@@@

@BEG_Contents

@BEG_Func
@RT(17)FuncTreeContainer
0
@END_Func

@BEG_Const
@RT(18)ConstTreeContainer
1
@Var @RT(16)cMoveEndParallel @RT(0) @T @F @DT @RT(0) @RT(0) @T @T @UNKNOWN 0 @F
@F @F
@T
@BEG_Attrib
0 @RT(0) @RT(0)
@END_Attrib
1 1 @F @F @F @F

@END_Const

@BEG_Export

@BEG_Kind
@FUNCTION_BLOCK @RT(29)FBInterpreterCheckIsRightJoin @STRUCTURED_TEXT
@RT(0) @RT(0) @RT(0)
@END_Kind

@BEG_Dcl
@RT(16)DclTreeContainer
7
@Var @RT(11)odcSequence @RT(0) @T @T @DERIVED 0 @T @T @DT @RT(13)KODC_Sequence @RT(0) @T @T @UNKNOWN 0 @F
@F @F
@T
@BEG_Attrib
3 @RT(0) @RT(11)[col][line] @RT(0)
@END_Attrib
1 2 @F @F @F @F

@Var @RT(18)iColumnStartBranch @RT(0) @T @F @DT @RT(4)DINT @RT(0) @T @T @BASIC 0 @F
@F @F
@T
@BEG_Attrib
3 @RT(0) @RT(0) @RT(0)
@END_Attrib
1 1 @F @F @F @F

@Var @RT(5)iLine @RT(0) @T @F @DT @RT(4)DINT @RT(0) @T @T @BASIC 0 @F
@F @F
@T
@BEG_Attrib
3 @RT(0) @RT(0) @RT(0)
@END_Attrib
1 1 @F @F @F @F

@Var @RT(7)bIsJoin @RT(0) @T @F @DT @RT(4)BOOL @RT(0) @T @T @BASIC 0 @F
@F @F
@T
@BEG_Attrib
3 @RT(0) @RT(0) @RT(0)
@END_Attrib
1 3 @F @F @F @F

@Var @RT(6)bError @RT(0) @T @F @DT @RT(4)BOOL @RT(0) @T @T @BASIC 0 @F
@F @F
@T
@BEG_Attrib
3 @RT(0) @RT(0) @RT(0)
@END_Attrib
1 3 @F @F @F @F

@Var @RT(10)iTmpColumn @RT(0) @T @F @DT @RT(4)DINT @RT(0) @T @T @BASIC 0 @F
@F @F
@T
@BEG_Attrib
3 @RT(0) @RT(0) @RT(0)
@END_Attrib
1 4 @F @F @F @F

@Var @RT(13)fbDebugTrace2 @RT(0) @T @T @DERIVED 0 @T @T @DT @RT(13)FBDebugTrace2 @RT(0) @T @T @UNKNOWN 0 @F
@F @F
@T
@BEG_Attrib
3 @RT(0) @RT(0) @RT(0)
@END_Attrib
1 0 @F @F @F @F

@END_Dcl

@END_Export

@BEG_Body
@TL(21)
bError := FALSE;
bIsJoin := FALSE;

FOR iTmpColumn := 1 TO cMaxParallelMovements DO
   IF odcSequence[iTmpColumn][iLine].iMoveId = cMoveEndParallel THEN
      IF iTmpColumn < iColumnStartBranch THEN
         fbDebugTrace2(nODCInterpreter, 'found a EndPParallel at pos:x/x, that tries to join to the wrong parent branch');
         bError := TRUE;
         RETURN; (* error tried to join to somewhere else
                  before we got our wanted join *)
      END_IF;
      IF iTmpColumn = iColumnStartBranch THEN
         (* found where this branch joins again with iColumn *)
         bIsJoin := TRUE;
         RETURN;
      END_IF;
      (* otherwise something else tries to join into this column from the right side
         this is OK, ignore it *)
   END_IF;
END_FOR;

@END_Body

@END_Contents
@@@BEG_Password@@@
NGhzZm9kYzQ=
@@@END_Password@@@

(* ---- FBInterpreterFindEndOfParallel.pu ---- *)
(*
@h    ! WARNING !
@h    The Kemro K2 system (including software) only meets category B according to EN 954-1,
@h    thus it is not intended for usage in safety-relevant control applications in the field
@h    of personal safety (e.g. emergency stop).
@h    To implement potentially necessary safety-relevant control tasks, always use additional
@h    external safety devices that are intended for the particular purpose, and meet the necessary
@h    functional safety.
@h    For further information see EN 954-1 (EN ISO 13849-1) and/or the K2-x00 user manual, chapter
@h    "CE conformity, directives and standards".

Find the end of a parallel branch in
*)

IMPORT_OVER_LISTFILE
 cMoveEndParallel
, FBInterpreterCheckIsRightJoin
, FBDebugTrace2
, KODC_Sequence

END_IMPORT

FUNCTION_BLOCK FBInterpreterFindEndOfParallel #DUMMY_EDIT_BLOCK

VAR_IN_OUT
 odcSequence : KODC_Sequence (* [col][line] *);
END_VAR

VAR_INPUT
 iColumn : DINT;
 iLine : DINT;
END_VAR

VAR_OUTPUT
 iMaxLineOfBranch : DINT;
END_VAR

VAR_TEMP
 i : DINT;
 k : DINT;
END_VAR

VAR
 fbInterpreterCheckIsRightJoin : FBInterpreterCheckIsRightJoin;
 fbDebugTrace2 : FBDebugTrace2;
END_VAR
#BEGIN_EDIT_BLOCK

(* col/line  point to a SP (leftmost of them)*)

iMaxLineOfBranch := 0;

FOR i := 1 TO cMaxParallelMovements DO
   IF odcSequence[i][iLine].iMoveId = cMoveStartParallel THEN
      IF i < iColumn THEN
         fbDebugTrace2(nODCInterpreter, 'error block called wrong iColumn must be the leftmost SP');
         RETURN;
      ELSIF i > iColumn THEN
         (* iColumn itself is skipped since it's join point is the same as at least another join point*)
         FOR k := iLine + 1 TO cMaxODCSteps DO
            IF odcSequence[i][k].iMoveId = cMoveEndParallel THEN
               (* now look to the left if the left most column is
               the same where the parallel branch started *)
               fbInterpreterCheckIsRightJoin(odcSequence := odcSequence, iColumnStartBranch := iColumn, iLine := k);
               IF fbInterpreterCheckIsRightJoin.bIsJoin THEN
                  iMaxLineOfBranch := MAX(iMaxLineOfBranch, k);
                  EXIT;
               END_IF;
               IF fbInterpreterCheckIsRightJoin.bError THEN
                  (* error printed inside the block already *)
                  iMaxLineOfBranch := 0;
                  RETURN;
               END_IF;
            END_IF;
         END_FOR;
      END_IF; // i < iColumn
   END_IF; // odcSequence[i][iLine].iMoveId = cMoveStartParallel
END_FOR;

IF iMaxLineOfBranch = 0 THEN
   fbDebugTrace2(nODCInterpreter, 'no branch join point found????');
   (* error no branch join point found for this branch?? *)
   RETURN;
END_IF;

;#END_EDIT_BLOCK END_FUNCTION_BLOCK

#END_OF_IEC_PART

@Puma @IecEditor 6 95 @Pou 25
@@@BEG_Comment@@@
@h    ! WARNING !
@h    The Kemro K2 system (including software) only meets category B according to EN 954-1,
@h    thus it is not intended for usage in safety-relevant control applications in the field
@h    of personal safety (e.g. emergency stop).
@h    To implement potentially necessary safety-relevant control tasks, always use additional
@h    external safety devices that are intended for the particular purpose, and meet the necessary
@h    functional safety.
@h    For further information see EN 954-1 (EN ISO 13849-1) and/or the K2-x00 user manual, chapter
@h    "CE conformity, directives and standards".

Find the end of a parallel branch in
@@@END_Comment@@@

@BEG_Contents

@BEG_Func
@RT(17)FuncTreeContainer
0
@END_Func

@BEG_Const
@RT(18)ConstTreeContainer
1
@Var @RT(16)cMoveEndParallel @RT(0) @T @F @DT @RT(0) @RT(0) @T @T @UNKNOWN 0 @F
@F @F
@T
@BEG_Attrib
0 @RT(0) @RT(0)
@END_Attrib
1 1 @F @F @F @F

@END_Const

@BEG_Export

@BEG_Kind
@FUNCTION_BLOCK @RT(30)FBInterpreterFindEndOfParallel @STRUCTURED_TEXT
@RT(0) @RT(0) @RT(0)
@END_Kind

@BEG_Dcl
@RT(16)DclTreeContainer
8
@Var @RT(29)fbInterpreterCheckIsRightJoin @RT(0) @T @T @DERIVED 0 @T @T @DT @RT(29)FBInterpreterCheckIsRightJoin @RT(0) @T @T @UNKNOWN 0 @F
@F @F
@T
@BEG_Attrib
3 @RT(0) @RT(0) @RT(0)
@END_Attrib
1 0 @F @F @F @F

@Var @RT(13)fbDebugTrace2 @RT(0) @T @T @DERIVED 0 @T @T @DT @RT(13)FBDebugTrace2 @RT(0) @T @T @UNKNOWN 0 @F
@F @F
@T
@BEG_Attrib
3 @RT(0) @RT(0) @RT(0)
@END_Attrib
1 0 @F @F @F @F

@Var @RT(11)odcSequence @RT(0) @T @T @DERIVED 0 @T @T @DT @RT(13)KODC_Sequence @RT(0) @T @T @UNKNOWN 0 @F
@F @F
@T
@BEG_Attrib
3 @RT(0) @RT(11)[col][line] @RT(0)
@END_Attrib
1 2 @F @F @F @F

@Var @RT(7)iColumn @RT(0) @T @F @DT @RT(4)DINT @RT(0) @T @T @BASIC 0 @F
@F @F
@T
@BEG_Attrib
3 @RT(0) @RT(0) @RT(0)
@END_Attrib
1 1 @F @F @F @F

@Var @RT(5)iLine @RT(0) @T @F @DT @RT(4)DINT @RT(0) @T @T @BASIC 0 @F
@F @F
@T
@BEG_Attrib
3 @RT(0) @RT(0) @RT(0)
@END_Attrib
1 1 @F @F @F @F

@Var @RT(16)iMaxLineOfBranch @RT(0) @T @F @DT @RT(4)DINT @RT(0) @T @T @BASIC 0 @F
@F @F
@T
@BEG_Attrib
3 @RT(0) @RT(0) @RT(0)
@END_Attrib
1 3 @F @F @F @F

@Var @RT(1)i @RT(0) @T @F @DT @RT(4)DINT @RT(0) @T @T @BASIC 0 @F
@F @F
@T
@BEG_Attrib
3 @RT(0) @RT(0) @RT(0)
@END_Attrib
1 4 @F @F @F @F

@Var @RT(1)k @RT(0) @T @F @DT @RT(4)DINT @RT(0) @T @T @BASIC 0 @F
@F @F
@T
@BEG_Attrib
3 @RT(0) @RT(0) @RT(0)
@END_Attrib
1 4 @F @F @F @F

@END_Dcl

@END_Export

@BEG_Body
@TL(39)

(* col/line  point to a SP (leftmost of them)*)

iMaxLineOfBranch := 0;

FOR i := 1 TO cMaxParallelMovements DO
   IF odcSequence[i][iLine].iMoveId = cMoveStartParallel THEN
      IF i < iColumn THEN
         fbDebugTrace2(nODCInterpreter, 'error block called wrong iColumn must be the leftmost SP');
         RETURN;
      ELSIF i > iColumn THEN
         (* iColumn itself is skipped since it's join point is the same as at least another join point*)
         FOR k := iLine + 1 TO cMaxODCSteps DO
            IF odcSequence[i][k].iMoveId = cMoveEndParallel THEN
               (* now look to the left if the left most column is
               the same where the parallel branch started *)
               fbInterpreterCheckIsRightJoin(odcSequence := odcSequence, iColumnStartBranch := iColumn, iLine := k);
               IF fbInterpreterCheckIsRightJoin.bIsJoin THEN
                  iMaxLineOfBranch := MAX(iMaxLineOfBranch, k);
                  EXIT;
               END_IF;
               IF fbInterpreterCheckIsRightJoin.bError THEN
                  (* error printed inside the block already *)
                  iMaxLineOfBranch := 0;
                  RETURN;
               END_IF;
            END_IF;
         END_FOR;
      END_IF; // i < iColumn
   END_IF; // odcSequence[i][iLine].iMoveId = cMoveStartParallel
END_FOR;

IF iMaxLineOfBranch = 0 THEN
   fbDebugTrace2(nODCInterpreter, 'no branch join point found????');
   (* error no branch join point found for this branch?? *)
   RETURN;
END_IF;

@END_Body

@END_Contents
@@@BEG_Password@@@
NGhzZm9kYzQ=
@@@END_Password@@@

(* ---- FBMoveDescription.pu ---- *)
IMPORT_OVER_LISTFILE
 tyMovementRegisterList
, tsODCDeviceMovementList

END_IMPORT

FUNCTION_BLOCK FBMoveDescription #DUMMY_EDIT_BLOCK

VAR_OUTPUT
 sDescription : STRING(255);
END_VAR

VAR_INPUT
 iMoveNr : DINT;
END_VAR

SYSTEM_VAR
 sv_MovementsAvailable : tyMovementRegisterList;
 sv_ODCDeviceMovements : tsODCDeviceMovementList;
END_VAR
#BEGIN_EDIT_BLOCK
(**************************************** WARNING ********************************************
 *** The KEBA Kemro K2 System including software is not intended for safety control tasks! ***
 ***                       For further information see Comment tab!                        ***
 *********************************************************************************************)

sDescription := CONCAT(sv_ODCDeviceMovements.Devices[sv_MovementsAvailable[iMoveNr].iFuIndex].sFuName,
                       " ",
                       sv_MovementsAvailable[iMoveNr].pMovementData^.sMoveId);

;#END_EDIT_BLOCK END_FUNCTION_BLOCK

#END_OF_IEC_PART

@Puma @IecEditor 6 96 @Pou 25
@@@BEG_Comment@@@

@@@END_Comment@@@

@BEG_Contents

@BEG_Func
@RT(17)FuncTreeContainer
0
@END_Func

@BEG_Const
@RT(18)ConstTreeContainer
0
@END_Const

@BEG_Export

@BEG_Kind
@FUNCTION_BLOCK @RT(17)FBMoveDescription @STRUCTURED_TEXT
@RT(0) @RT(0) @RT(0)
@END_Kind

@BEG_Dcl
@RT(16)DclTreeContainer
4
@Var @RT(12)sDescription @RT(0) @T @F @DT @RT(11)STRING(255) @RT(0) @T @T @STRING 0 @F @RT(3)255 @F
@F @F
@T
@BEG_Attrib
3 @RT(0) @RT(0) @RT(0)
@END_Attrib
1 3 @F @F @F @F

@Var @RT(7)iMoveNr @RT(0) @T @F @DT @RT(4)DINT @RT(0) @T @T @BASIC 0 @F
@F @F
@T
@BEG_Attrib
3 @RT(0) @RT(0) @RT(0)
@END_Attrib
1 1 @F @F @F @F

@Var @RT(21)sv_MovementsAvailable @RT(0) @T @T @DERIVED 0 @T @T @DT @RT(22)tyMovementRegisterList @RT(0) @T @T @UNKNOWN 0 @F
@F @F
@T
@BEG_Attrib
3 @RT(0) @RT(0) @RT(0)
@END_Attrib
1 8 @F @F @F @F

@Var @RT(21)sv_ODCDeviceMovements @RT(0) @T @T @RENAMED 0 @T @T @DT @RT(23)tsODCDeviceMovementList @RT(0) @T @T @UNKNOWN 0 @F
@F @F
@T
@BEG_Attrib
3 @RT(0) @RT(0) @RT(0)
@END_Attrib
1 8 @F @F @F @F

@END_Dcl

@END_Export

@BEG_Body
@TL(11)
(**************************************** WARNING ********************************************
 *** The KEBA Kemro K2 System including software is not intended for safety control tasks! ***
 ***                       For further information see Comment tab!                        ***
 *********************************************************************************************)

sDescription := CONCAT(sv_ODCDeviceMovements.Devices[sv_MovementsAvailable[iMoveNr].iFuIndex].sFuName,
                       " ",
                       sv_MovementsAvailable[iMoveNr].pMovementData^.sMoveId);

@END_Body

@END_Contents
@@@BEG_Password@@@
NGhzZm9kYzQ=
@@@END_Password@@@

(* ---- FBSetStepState.pu ---- *)
(*
Update the current state of a step to the internal ODC sequence array
at sv_ODCSequenceInt.StepState

This state is used on the HMI to display errors, the currently executing step
and finished steps.
*)

IMPORT_OVER_LISTFILE
 tyODCSequenceInternal
, tsODCStepPos
, tnODCStepState

END_IMPORT

FUNCTION_BLOCK FBSetStepState #DUMMY_EDIT_BLOCK

VAR_INPUT
 StepPos : tsODCStepPos (* Position of the step for which to update the state *);
 StepState : tnODCStepState (* New state *);
END_VAR

SYSTEM_VAR
 sv_ODCSequenceInt : tyODCSequenceInternal;
END_VAR
#BEGIN_EDIT_BLOCK
(**************************************** WARNING ********************************************
 *** The KEBA Kemro K2 System including software is not intended for safety control tasks! ***
 ***                       For further information see Comment tab!                        ***
 *********************************************************************************************)

sv_ODCSequenceInt[StepPos.iColumn][StepPos.iRow].StepState := StepState;

sv_ODCSequenceInt[StepPos.iColumn][StepPos.iRow].bStepActive := (StepState = nStateActive);
sv_ODCSequenceInt[StepPos.iColumn][StepPos.iRow].bStepDone := (StepState = nStateReady);

;#END_EDIT_BLOCK END_FUNCTION_BLOCK

#END_OF_IEC_PART

@Puma @IecEditor 6 96 @Pou 25
@@@BEG_Comment@@@
Update the current state of a step to the internal ODC sequence array
at sv_ODCSequenceInt.StepState

This state is used on the HMI to display errors, the currently executing step
and finished steps.
@@@END_Comment@@@

@BEG_Contents

@BEG_Func
@RT(17)FuncTreeContainer
0
@END_Func

@BEG_Const
@RT(18)ConstTreeContainer
0
@END_Const

@BEG_Export

@BEG_Kind
@FUNCTION_BLOCK @RT(14)FBSetStepState @STRUCTURED_TEXT
@RT(0) @RT(0) @RT(0)
@END_Kind

@BEG_Dcl
@RT(16)DclTreeContainer
3
@Var @RT(17)sv_ODCSequenceInt @RT(0) @T @T @DERIVED 0 @F @RT(21)tyODCSequenceInternal @F
@T
@BEG_Attrib
3 @RT(0) @RT(0) @RT(0)
@END_Attrib
1 8 @F @F @F @F

@Var @RT(7)StepPos @RT(0) @T @T @DERIVED 0 @T @T @DT @RT(12)tsODCStepPos @RT(0) @T @T @UNKNOWN 0 @F
@F @F
@T
@BEG_Attrib
3 @RT(0) @RT(50)Position of the step for which to update the state @RT(0)
@END_Attrib
1 1 @F @F @F @F

@Var @RT(9)StepState @RT(0) @T @T @DERIVED 0 @T @T @DT @RT(14)tnODCStepState @RT(0) @T @T @UNKNOWN 0 @F
@F @F
@T
@BEG_Attrib
3 @RT(0) @RT(9)New state @RT(0)
@END_Attrib
1 1 @F @F @F @F

@END_Dcl

@END_Export

@BEG_Body
@TL(10)
(**************************************** WARNING ********************************************
 *** The KEBA Kemro K2 System including software is not intended for safety control tasks! ***
 ***                       For further information see Comment tab!                        ***
 *********************************************************************************************)

sv_ODCSequenceInt[StepPos.iColumn][StepPos.iRow].StepState := StepState;

sv_ODCSequenceInt[StepPos.iColumn][StepPos.iRow].bStepActive := (StepState = nStateActive);
sv_ODCSequenceInt[StepPos.iColumn][StepPos.iRow].bStepDone := (StepState = nStateReady);

@END_Body

@END_Contents
@@@BEG_Password@@@
NGhzZm9kYzQ=
@@@END_Password@@@

(* ---- FBStartedMovementAdder.pu ---- *)
(*
@h    ! WARNING !
@h    The Kemro K2 system (including software) only meets category B according to EN 954-1,
@h    thus it is not intended for usage in safety-relevant control applications in the field
@h    of personal safety (e.g. emergency stop).
@h    To implement potentially necessary safety-relevant control tasks, always use additional
@h    external safety devices that are intended for the particular purpose, and meet the necessary
@h    functional safety.
@h    For further information see EN 954-1 (EN ISO 13849-1) and/or the K2-x00 user manual, chapter
@h    "CE conformity, directives and standards".
*)

IMPORT_OVER_LISTFILE
 SET_ALARM
, ASSERT
, cMaxActiveMovements
, tsDeviceId
, tsODCStepPos
, tMoveIdent
, tsStartedMoveDataODCExtended
, KRTOS_Semaphore
, KRTOS_Status
, tsTraceLevel

END_IMPORT

FUNCTION_BLOCK FBStartedMovementAdder #DUMMY_EDIT_BLOCK

VAR_INPUT
 DeviceId : tsDeviceId;
 StepPos : tsODCStepPos;
 MoveId : tMoveIdent;
 MoveDir : tMoveIdent;
 iInstance : DINT;
END_VAR

VAR_OUTPUT
 bOK : BOOL;
END_VAR

SYSTEM_VAR
 sv_StartedManualMovements : tsStartedMoveDataODCExtended;
 sv_TraceLevel : tsTraceLevel;
END_VAR

SYSTEM_OBJECT
 erMaxStartedMovementsExceeded : ALARM;
 erAssert : ALARM;
END_OBJECT

VAR_EXTERNAL
 MovementsSema : KRTOS_Semaphore (* protects sv_StartedManualMovements *);
END_VAR

VAR_TEMP
 i : DINT;
END_VAR

VAR
 dummy : DINT;
 dummy2 : BOOL;
 Status : KRTOS_Status;
END_VAR
#BEGIN_EDIT_BLOCK
(**************************************** WARNING ********************************************
 *** The KEBA Kemro K2 System including software is not intended for safety control tasks! ***
 ***                       For further information see Comment tab!                        ***
 *********************************************************************************************)

bOK := FALSE;

Status := MovementsSema.Wait(WaitTime := cTimeOutSempahore);
IF Status <> KRTOS_Status_OK THEN
   dummy2 := ASSERT(FALSE, erAssert);
   RETURN;
END_IF;

IF sv_StartedManualMovements.iStartedMovements < cMaxActiveMovements THEN
   //add movement to sv_StartedManualMovements
   IF sv_TraceLevel.bODCInterpreter THEN
      dummy := Print('adding started manual movement %d.%d %d/%d pos: %d/%d', DeviceId.CompId, DeviceId.IndexId, MoveId, MoveDir, StepPos.iColumn, StepPos.iRow);
   END_IF;

   sv_StartedManualMovements.iStartedMovements := sv_StartedManualMovements.iStartedMovements +1;
   sv_StartedManualMovements.MoveData[sv_StartedManualMovements.iStartedMovements].DeviceId := DeviceId;
   sv_StartedManualMovements.MoveData[sv_StartedManualMovements.iStartedMovements].MoveDir := MoveDir;
   sv_StartedManualMovements.MoveData[sv_StartedManualMovements.iStartedMovements].MoveId := MoveId;
   sv_StartedManualMovements.MoveData[sv_StartedManualMovements.iStartedMovements].StepPos := StepPos;
   sv_StartedManualMovements.MoveData[sv_StartedManualMovements.iStartedMovements].iInstance := iInstance;
   bOK := TRUE;
ELSE
   //too many movements started
   //show some information about the movement to make debugging easier
   dummy := Print('set alarm erMaxStartedMovementsExceeded in FBStartedMovementAdder.pu');
   dummy := Print('max. active movements: %d', cMaxActiveMovements);
   dummy := Print('tried to start    %d.%d %d/%d',
                  DeviceId.CompId, DeviceId.IndexId,
                  MoveId, MoveDir);
   FOR i := 1 TO cMaxActiveMovements DO
      dummy := Print('already started %d %d.%d %d/%d',
                     i, sv_StartedManualMovements.MoveData[i].DeviceId.CompId, sv_StartedManualMovements.MoveData[i].DeviceId.IndexId,
                     sv_StartedManualMovements.MoveData[i].MoveId, sv_StartedManualMovements.MoveData[i].MoveDir);
   END_FOR;
   //set alarm after tracing out
   SET_ALARM(Name := erMaxStartedMovementsExceeded,
            SubID1 := cMaxActiveMovements);
END_IF;

Status := MovementsSema.Put();
IF Status <> KRTOS_Status_OK THEN
   dummy2 := ASSERT(FALSE, erAssert);
END_IF;

;#END_EDIT_BLOCK END_FUNCTION_BLOCK

#END_OF_IEC_PART

@Puma @IecEditor 6 96 @Pou 25
@@@BEG_Comment@@@
@h    ! WARNING !
@h    The Kemro K2 system (including software) only meets category B according to EN 954-1,
@h    thus it is not intended for usage in safety-relevant control applications in the field
@h    of personal safety (e.g. emergency stop).
@h    To implement potentially necessary safety-relevant control tasks, always use additional
@h    external safety devices that are intended for the particular purpose, and meet the necessary
@h    functional safety.
@h    For further information see EN 954-1 (EN ISO 13849-1) and/or the K2-x00 user manual, chapter
@h    "CE conformity, directives and standards".
@@@END_Comment@@@

@BEG_Contents

@BEG_Func
@RT(17)FuncTreeContainer
2
@Var @RT(9)SET_ALARM @RT(0) @T @T @DERIVED 0 @F @RT(23)KEBA_STANDARD_PROCEDURE @F
@T
@BEG_Attrib
0 @RT(0) @RT(0)
@END_Attrib
1 1 @F @F @F @F

@Var @RT(6)ASSERT @RT(0) @T @T @DERIVED 0 @F @RT(8)FUNCTION @F
@T
@BEG_Attrib
0 @RT(0) @RT(0)
@END_Attrib
1 1 @F @F @F @F

@END_Func

@BEG_Const
@RT(18)ConstTreeContainer
1
@Var @RT(19)cMaxActiveMovements @RT(0) @T @F @DT @RT(4)DINT @RT(0) @T @T @BASIC 0 @F
@F @F
@T
@BEG_Attrib
0 @RT(1)6 @RT(52)number of movements that are active at the same time
@END_Attrib
1 1 @F @F @F @F

@END_Const

@BEG_Export

@BEG_Kind
@FUNCTION_BLOCK @RT(22)FBStartedMovementAdder @STRUCTURED_TEXT
@RT(0) @RT(0) @RT(0)
@END_Kind

@BEG_Dcl
@RT(16)DclTreeContainer
15
@Var @RT(8)DeviceId @RT(0) @T @T @DERIVED 0 @T @T @DT @RT(10)tsDeviceId @RT(0) @T @T @UNKNOWN 0 @F
@F @F
@T
@BEG_Attrib
3 @RT(0) @RT(0) @RT(0)
@END_Attrib
1 1 @F @F @F @F

@Var @RT(7)StepPos @RT(0) @T @T @DERIVED 0 @F @RT(12)tsODCStepPos @F
@T
@BEG_Attrib
3 @RT(0) @RT(0) @RT(0)
@END_Attrib
1 1 @F @F @F @F

@Var @RT(6)MoveId @RT(0) @T @T @DERIVED 0 @T @T @DT @RT(10)tMoveIdent @RT(0) @T @T @UNKNOWN 0 @F
@F @F
@T
@BEG_Attrib
3 @RT(0) @RT(0) @RT(0)
@END_Attrib
1 1 @F @F @F @F

@Var @RT(7)MoveDir @RT(0) @T @T @DERIVED 0 @T @T @DT @RT(10)tMoveIdent @RT(0) @T @T @UNKNOWN 0 @F
@F @F
@T
@BEG_Attrib
3 @RT(0) @RT(0) @RT(0)
@END_Attrib
1 1 @F @F @F @F

@Var @RT(9)iInstance @RT(0) @T @F @DT @RT(4)DINT @RT(0) @T @T @BASIC 0 @F
@F @F
@T
@BEG_Attrib
3 @RT(0) @RT(0) @RT(0)
@END_Attrib
1 1 @F @F @F @F

@Var @RT(3)bOK @RT(0) @T @F @DT @RT(4)BOOL @RT(0) @T @T @BASIC 0 @F
@F @F
@T
@BEG_Attrib
3 @RT(0) @RT(0) @RT(0)
@END_Attrib
1 3 @F @F @F @F

@Var @RT(25)sv_StartedManualMovements @RT(0) @T @T @RENAMED 0 @T @T @DT @RT(28)tsStartedMoveDataODCExtended @RT(0) @T @T @UNKNOWN 0 @F
@F @F
@T
@BEG_Attrib
3 @RT(0) @RT(0) @RT(0)
@END_Attrib
1 8 @F @F @F @F

@Var @RT(29)erMaxStartedMovementsExceeded @RT(0) @T @T @RENAMED 0 @T @T @DT @RT(5)ALARM @RT(0) @T @T @BASIC 0 @F
@F @F
@T
@BEG_Attrib
3 @RT(0) @RT(0) @RT(0)
@END_Attrib
1 7 @F @F @F @F

@Var @RT(8)erAssert @RT(0) @T @T @RENAMED 0 @T @T @DT @RT(5)ALARM @RT(0) @T @T @BASIC 0 @F
@F @F
@T
@BEG_Attrib
3 @RT(0) @RT(0) @RT(0)
@END_Attrib
1 7 @F @F @F @F

@Var @RT(13)MovementsSema @RT(0) @T @T @DERIVED 0 @T @T @DT @RT(15)KRTOS_Semaphore @RT(0) @T @T @UNKNOWN 0 @F
@F @F
@T
@BEG_Attrib
3 @RT(0) @RT(34)protects sv_StartedManualMovements @RT(0)
@END_Attrib
1 6 @F @F @F @F

@Var @RT(5)dummy @RT(0) @T @F @DT @RT(4)DINT @RT(0) @T @T @BASIC 0 @F
@F @F
@T
@BEG_Attrib
3 @RT(0) @RT(0) @RT(0)
@END_Attrib
1 0 @F @F @F @F

@Var @RT(6)dummy2 @RT(0) @T @F @DT @RT(4)BOOL @RT(0) @T @T @BASIC 0 @F
@F @F
@T
@BEG_Attrib
3 @RT(0) @RT(0) @RT(0)
@END_Attrib
1 0 @F @F @F @F

@Var @RT(6)Status @RT(0) @T @T @DERIVED 0 @T @T @DT @RT(12)KRTOS_Status @RT(0) @T @T @UNKNOWN 0 @F
@F @F
@T
@BEG_Attrib
3 @RT(0) @RT(0) @RT(0)
@END_Attrib
1 0 @F @F @F @F

@Var @RT(13)sv_TraceLevel @RT(0) @T @T @DERIVED 0 @T @T @DT @RT(12)tsTraceLevel @RT(0) @T @T @UNKNOWN 0 @F
@F @F
@T
@BEG_Attrib
3 @RT(0) @RT(0) @RT(0)
@END_Attrib
1 8 @F @F @F @F

@Var @RT(1)i @RT(0) @T @F @DT @RT(4)DINT @RT(0) @T @T @BASIC 0 @F
@F @F
@T
@BEG_Attrib
3 @RT(0) @RT(0) @RT(0)
@END_Attrib
1 4 @F @F @F @F

@END_Dcl

@END_Export

@BEG_Body
@TL(49)
(**************************************** WARNING ********************************************
 *** The KEBA Kemro K2 System including software is not intended for safety control tasks! ***
 ***                       For further information see Comment tab!                        ***
 *********************************************************************************************)

bOK := FALSE;

Status := MovementsSema.Wait(WaitTime := cTimeOutSempahore);
IF Status <> KRTOS_Status_OK THEN
   dummy2 := ASSERT(FALSE, erAssert);
   RETURN;
END_IF;

IF sv_StartedManualMovements.iStartedMovements < cMaxActiveMovements THEN
   //add movement to sv_StartedManualMovements
   IF sv_TraceLevel.bODCInterpreter THEN
      dummy := Print('adding started manual movement %d.%d %d/%d pos: %d/%d', DeviceId.CompId, DeviceId.IndexId, MoveId, MoveDir, StepPos.iColumn, StepPos.iRow);
   END_IF;

   sv_StartedManualMovements.iStartedMovements := sv_StartedManualMovements.iStartedMovements +1;
   sv_StartedManualMovements.MoveData[sv_StartedManualMovements.iStartedMovements].DeviceId := DeviceId;
   sv_StartedManualMovements.MoveData[sv_StartedManualMovements.iStartedMovements].MoveDir := MoveDir;
   sv_StartedManualMovements.MoveData[sv_StartedManualMovements.iStartedMovements].MoveId := MoveId;
   sv_StartedManualMovements.MoveData[sv_StartedManualMovements.iStartedMovements].StepPos := StepPos;
   sv_StartedManualMovements.MoveData[sv_StartedManualMovements.iStartedMovements].iInstance := iInstance;
   bOK := TRUE;
ELSE
   //too many movements started
   //show some information about the movement to make debugging easier
   dummy := Print('set alarm erMaxStartedMovementsExceeded in FBStartedMovementAdder.pu');
   dummy := Print('max. active movements: %d', cMaxActiveMovements);
   dummy := Print('tried to start    %d.%d %d/%d',
                  DeviceId.CompId, DeviceId.IndexId,
                  MoveId, MoveDir);
   FOR i := 1 TO cMaxActiveMovements DO
      dummy := Print('already started %d %d.%d %d/%d',
                     i, sv_StartedManualMovements.MoveData[i].DeviceId.CompId, sv_StartedManualMovements.MoveData[i].DeviceId.IndexId,
                     sv_StartedManualMovements.MoveData[i].MoveId, sv_StartedManualMovements.MoveData[i].MoveDir);
   END_FOR;
   //set alarm after tracing out
   SET_ALARM(Name := erMaxStartedMovementsExceeded,
            SubID1 := cMaxActiveMovements);
END_IF;

Status := MovementsSema.Put();
IF Status <> KRTOS_Status_OK THEN
   dummy2 := ASSERT(FALSE, erAssert);
END_IF;

@END_Body

@END_Contents
@@@BEG_Password@@@
NGhzZm9kYzQ=
@@@END_Password@@@

(* ---- FBStopStartedManualMovements.pu ---- *)
(*
@h    ! WARNING !
@h    The Kemro K2 system (including software) only meets category B according to EN 954-1,
@h    thus it is not intended for usage in safety-relevant control applications in the field
@h    of personal safety (e.g. emergency stop).
@h    To implement potentially necessary safety-relevant control tasks, always use additional
@h    external safety devices that are intended for the particular purpose, and meet the necessary
@h    functional safety.
@h    For further information see EN 954-1 (EN ISO 13849-1) and/or the K2-x00 user manual, chapter
@h    "CE conformity, directives and standards".

*)

IMPORT_OVER_LISTFILE
 tsStartedMoveDataODCExtended
, FBDebugTrace2
, FBStop

END_IMPORT

FUNCTION_BLOCK FBStopStartedManualMovements #DUMMY_EDIT_BLOCK

SYSTEM_VAR
 sv_StartedManualMovements : tsStartedMoveDataODCExtended;
END_VAR

VAR_TEMP
 i : DINT;
END_VAR

VAR
 StartedMovements : tsStartedMoveDataODCExtended;
 fbDebugTrace2 : FBDebugTrace2;
 fbStop : FBStop;
END_VAR
#BEGIN_EDIT_BLOCK
(**************************************** WARNING ********************************************
 *** The KEBA Kemro K2 System including software is not intended for safety control tasks! ***
 ***                       For further information see Comment tab!                        ***
 *********************************************************************************************)

//copy systemvariable to local variable because systemvariable can be changed during executing the code
fbDebugTrace2(nDeviceState, 'stopping all started manual movements');
StartedMovements := sv_StartedManualMovements;

FOR i := 1 TO StartedMovements.iStartedMovements DO
   //stop all started movements
   fbDebugTrace2(nDeviceState, CONCAT('FBStopStartedManualMovements.pu stopping device ',
                 DINT_TO_STRING(StartedMovements.MoveData[i].DeviceId.CompId),
                 '/',
                 DINT_TO_STRING(StartedMovements.MoveData[i].DeviceId.IndexId),
                 ' (list entry ',
                 DINT_TO_STRING(i),
                 ' of ',
                 DINT_TO_STRING(StartedMovements.iStartedMovements),
                 ')'));
   fbStop(DeviceId := StartedMovements.MoveData[i].DeviceId);
END_FOR;

;#END_EDIT_BLOCK END_FUNCTION_BLOCK

#END_OF_IEC_PART

@Puma @IecEditor 6 96 @Pou 25
@@@BEG_Comment@@@
@h    ! WARNING !
@h    The Kemro K2 system (including software) only meets category B according to EN 954-1,
@h    thus it is not intended for usage in safety-relevant control applications in the field
@h    of personal safety (e.g. emergency stop).
@h    To implement potentially necessary safety-relevant control tasks, always use additional
@h    external safety devices that are intended for the particular purpose, and meet the necessary
@h    functional safety.
@h    For further information see EN 954-1 (EN ISO 13849-1) and/or the K2-x00 user manual, chapter
@h    "CE conformity, directives and standards".

@@@END_Comment@@@

@BEG_Contents

@BEG_Func
@RT(17)FuncTreeContainer
0
@END_Func

@BEG_Const
@RT(18)ConstTreeContainer
0
@END_Const

@BEG_Export

@BEG_Kind
@FUNCTION_BLOCK @RT(28)FBStopStartedManualMovements @STRUCTURED_TEXT
@RT(0) @RT(0) @RT(0)
@END_Kind

@BEG_Dcl
@RT(16)DclTreeContainer
5
@Var @RT(25)sv_StartedManualMovements @RT(0) @T @T @DERIVED 0 @T @T @DT @RT(28)tsStartedMoveDataODCExtended @RT(0) @T @T @UNKNOWN 0 @F
@F @F
@T
@BEG_Attrib
3 @RT(0) @RT(0) @RT(0)
@END_Attrib
1 8 @F @F @F @F

@Var @RT(16)StartedMovements @RT(0) @T @T @DERIVED 0 @T @T @DT @RT(28)tsStartedMoveDataODCExtended @RT(0) @T @T @UNKNOWN 0 @F
@F @F
@T
@BEG_Attrib
3 @RT(0) @RT(0) @RT(0)
@END_Attrib
1 0 @F @F @F @F

@Var @RT(13)fbDebugTrace2 @RT(0) @T @T @DERIVED 0 @T @T @DT @RT(13)FBDebugTrace2 @RT(0) @T @T @UNKNOWN 0 @F
@F @F
@T
@BEG_Attrib
3 @RT(0) @RT(0) @RT(0)
@END_Attrib
1 0 @F @F @F @F

@Var @RT(6)fbStop @RT(0) @T @T @DERIVED 0 @T @T @DT @RT(6)FBStop @RT(0) @T @T @UNKNOWN 0 @F
@F @F
@T
@BEG_Attrib
3 @RT(0) @RT(0) @RT(0)
@END_Attrib
1 0 @F @F @F @F

@Var @RT(1)i @RT(0) @T @F @DT @RT(4)DINT @RT(0) @T @T @BASIC 0 @F
@F @F
@T
@BEG_Attrib
3 @RT(0) @RT(0) @RT(0)
@END_Attrib
1 4 @F @F @F @F

@END_Dcl

@END_Export

@BEG_Body
@TL(24)
(**************************************** WARNING ********************************************
 *** The KEBA Kemro K2 System including software is not intended for safety control tasks! ***
 ***                       For further information see Comment tab!                        ***
 *********************************************************************************************)

//copy systemvariable to local variable because systemvariable can be changed during executing the code
fbDebugTrace2(nDeviceState, 'stopping all started manual movements');
StartedMovements := sv_StartedManualMovements;

FOR i := 1 TO StartedMovements.iStartedMovements DO
   //stop all started movements
   fbDebugTrace2(nDeviceState, CONCAT('FBStopStartedManualMovements.pu stopping device ',
                 DINT_TO_STRING(StartedMovements.MoveData[i].DeviceId.CompId),
                 '/',
                 DINT_TO_STRING(StartedMovements.MoveData[i].DeviceId.IndexId),
                 ' (list entry ',
                 DINT_TO_STRING(i),
                 ' of ',
                 DINT_TO_STRING(StartedMovements.iStartedMovements),
                 ')'));
   fbStop(DeviceId := StartedMovements.MoveData[i].DeviceId);
END_FOR;

@END_Body

@END_Contents
@@@BEG_Password@@@
NGhzZm9kYzQ=
@@@END_Password@@@

(* ---- ABActiveGroups.pu ---- *)
(*
@h    ! WARNING !
@h    The Kemro K2 system (including software) only meets category B according to EN 954-1,
@h    thus it is not intended for usage in safety-relevant control applications in the field
@h    of personal safety (e.g. emergency stop).
@h    To implement potentially necessary safety-relevant control tasks, always use additional
@h    external safety devices that are intended for the particular purpose, and meet the necessary
@h    functional safety.
@h    For further information see EN 954-1 (EN ISO 13849-1) and/or the K2-x00 user manual, chapter
@h    "CE conformity, directives and standards".

AB for maintenance of the active times of the programmed groups.
*)

IMPORT_OVER_LISTFILE
 STOP_PROCESS_ALGORITHM
, tyInterCondTimeArray
, tsGroupActiveData
, RTC

END_IMPORT

ALGORITHM_BLOCK ABActiveGroups #DUMMY_EDIT_BLOCK

SYSTEM_VAR
 sv_GroupActiveTimes : tyInterCondTimeArray (* array with act. times for all groups *);
 sv_GroupActiveData : tsGroupActiveData;
END_VAR

SYSTEM_OBJECT
 PU_Task_3 : TASK;
 TaskAnalog : TASK;
END_OBJECT

POSTUPDATE_ALGORITHM pActiveGroups ON PU_Task_3 WITH sv_GroupActiveData.iActiveGroups

#BEGIN_EDIT_BLOCK
(**************************************** WARNING ********************************************
 *** The KEBA Kemro K2 System including software is not intended for safety control tasks! ***
 ***                       For further information see Comment tab!                        ***
 *********************************************************************************************)

IF sv_GroupActiveData.iActiveGroups > 0 THEN
   START_PROCESS_ALGORITHM(paActiveGroupTimes);
ELSE
   STOP_PROCESS_ALGORITHM(paActiveGroupTimes);
END_IF;

;#END_EDIT_BLOCK END_ALGORITHM

PROCESS_ALGORITHM paActiveGroupTimes ON TaskAnalog

VAR_TEMP
 i : DINT;
END_VAR

VAR
 fbRTC : RTC;
 dActTime : DATE_AND_TIME;
END_VAR
#BEGIN_EDIT_BLOCK
(**************************************** WARNING ********************************************
 *** The KEBA Kemro K2 System including software is not intended for safety control tasks! ***
 ***                       For further information see Comment tab!                        ***
 *********************************************************************************************)

fbRTC();
dActTime := fbRTC.CDT;

FOR i := 1 TO cMaxIntermediateConditions DO
   IF sv_GroupActiveData.Group[i].bActive THEN
      sv_GroupActiveTimes[i] := (dActTime - sv_GroupActiveData.Group[i].dStartTime);
   END_IF;
END_FOR;

;#END_EDIT_BLOCK END_ALGORITHM

END_ALGORITHM_BLOCK

#END_OF_IEC_PART

@Puma @IecEditor 6 127 @Pou 25
@@@BEG_Comment@@@
@h    ! WARNING !
@h    The Kemro K2 system (including software) only meets category B according to EN 954-1,
@h    thus it is not intended for usage in safety-relevant control applications in the field
@h    of personal safety (e.g. emergency stop).
@h    To implement potentially necessary safety-relevant control tasks, always use additional
@h    external safety devices that are intended for the particular purpose, and meet the necessary
@h    functional safety.
@h    For further information see EN 954-1 (EN ISO 13849-1) and/or the K2-x00 user manual, chapter
@h    "CE conformity, directives and standards".

AB for maintenance of the active times of the programmed groups.
@@@END_Comment@@@

@BEG_Contents

@BEG_Func
@RT(17)FuncTreeContainer
1
@Var @RT(22)STOP_PROCESS_ALGORITHM @RT(0) @T @T @DERIVED 0 @F @RT(23)KEBA_STANDARD_PROCEDURE @F
@T
@BEG_Attrib
0 @RT(0) @RT(0)
@END_Attrib
1 1 @F @F @F @F

@END_Func

@BEG_Const
@RT(18)ConstTreeContainer
0
@END_Const

@BEG_Export

@BEG_Kind
@ALGORITHM_BLOCK @RT(14)ABActiveGroups @STRUCTURED_TEXT
@RT(0) @RT(0) @RT(0)
@END_Kind

@BEG_Dcl
@RT(16)DclTreeContainer
4
@Var @RT(19)sv_GroupActiveTimes @RT(0) @T @T @DERIVED 0 @T @T @DT @RT(20)tyInterCondTimeArray @RT(0) @T @T @UNKNOWN 0 @F
@F @F
@T
@BEG_Attrib
3 @RT(0) @RT(36)array with act. times for all groups @RT(0)
@END_Attrib
1 8 @F @F @F @F

@Var @RT(18)sv_GroupActiveData @RT(0) @T @T @DERIVED 0 @T @T @DT @RT(17)tsGroupActiveData @RT(0) @T @T @UNKNOWN 0 @F
@F @F
@T
@BEG_Attrib
3 @RT(0) @RT(0) @RT(0)
@END_Attrib
1 8 @F @F @F @F

@Var @RT(9)PU_Task_3 @RT(0) @T @T @RENAMED 0 @T @T @DT @RT(4)TASK @RT(0) @T @T @BASIC 0 @F
@F @F
@T
@BEG_Attrib
3 @RT(0) @RT(0) @RT(0)
@END_Attrib
1 7 @F @F @F @F

@Var @RT(10)TaskAnalog @RT(0) @T @T @RENAMED 0 @T @T @DT @RT(4)TASK @RT(0) @T @T @BASIC 0 @F
@F @F
@T
@BEG_Attrib
3 @RT(0) @RT(0) @RT(0)
@END_Attrib
1 7 @F @F @F @F

@END_Dcl

@END_Export

@BEG_Body

2

@BEG_Export

@BEG_Algo
@POSTUPDATE_ALGORITHM @RT(13)pActiveGroups @STRUCTURED_TEXT
@RT(0) @RT(32)sv_GroupActiveData.iActiveGroups @RT(9)PU_Task_3 @F @F
@END_Algo

@BEG_Dcl
@RT(16)DclTreeContainer
0
@END_Dcl

@END_Export

@BEG_Export

@BEG_Algo
@PROCESS_ALGORITHM @RT(18)paActiveGroupTimes @STRUCTURED_TEXT
@RT(0) @RT(0) @RT(10)TaskAnalog @F @F
@END_Algo

@BEG_Dcl
@RT(16)DclTreeContainer
3
@Var @RT(5)fbRTC @RT(0) @T @T @DERIVED 0 @T @T @DT @RT(3)RTC @RT(0) @T @T @UNKNOWN 0 @F
@F @F
@T
@BEG_Attrib
3 @RT(0) @RT(0) @RT(0)
@END_Attrib
1 0 @F @F @F @F

@Var @RT(8)dActTime @RT(0) @T @F @DT @RT(13)DATE_AND_TIME @RT(0) @T @T @BASIC 0 @F
@F @F
@T
@BEG_Attrib
3 @RT(0) @RT(0) @RT(0)
@END_Attrib
1 0 @F @F @F @F

@Var @RT(1)i @RT(0) @T @F @DT @RT(4)DINT @RT(0) @T @T @BASIC 0 @F
@F @F
@T
@BEG_Attrib
3 @RT(0) @RT(0) @RT(0)
@END_Attrib
1 4 @F @F @F @F

@END_Dcl

@END_Export

@BEG_Body
@TL(11)
(**************************************** WARNING ********************************************
 *** The KEBA Kemro K2 System including software is not intended for safety control tasks! ***
 ***                       For further information see Comment tab!                        ***
 *********************************************************************************************)

IF sv_GroupActiveData.iActiveGroups > 0 THEN
   START_PROCESS_ALGORITHM(paActiveGroupTimes);
ELSE
   STOP_PROCESS_ALGORITHM(paActiveGroupTimes);
END_IF;

@END_Body

@@@BEG_Comment@@@
@TL(0)

@@@END_Comment@@@

@BEG_Body
@TL(14)
(**************************************** WARNING ********************************************
 *** The KEBA Kemro K2 System including software is not intended for safety control tasks! ***
 ***                       For further information see Comment tab!                        ***
 *********************************************************************************************)

fbRTC();
dActTime := fbRTC.CDT;

FOR i := 1 TO cMaxIntermediateConditions DO
   IF sv_GroupActiveData.Group[i].bActive THEN
      sv_GroupActiveTimes[i] := (dActTime - sv_GroupActiveData.Group[i].dStartTime);
   END_IF;
END_FOR;

@END_Body

@@@BEG_Comment@@@
@TL(0)

@@@END_Comment@@@
@END_Body

@END_Contents
